C01747=-28.112,-95.435,39.346,-179.6955,-1.2364,-6766.4132
C01748=-32.220,-94.603,39.491,179.9985,-0.0489,-6768.8079
C01749=-36.266,-93.184,39.587,-179.9979,-0.0053,-6771.2653
C01750=-40.247,-91.535,39.587,179.9971,-0.0076,-6773.7346
C01751=-44.111,-89.678,39.491,179.9997,-0.0512,-6776.1917
C01752=-47.604,-87.360,39.346,179.6949,-1.2364,-6778.5867
C01753=-50.060,-84.322,39.203,179.1149,-1.5518,-6780.6966
C01754=-51.116,-81.128,39.027,177.5559,-1.8116,-6782.2136
C01755=-50.704,-78.221,38.697,177.2195,-0.9491,-6782.9519
C01756=-49.835,-75.348,38.031,-179.8330,0.0487,-6783.4806
C01757=-49.130,-72.694,37.169,-173.6149,2.5069,-6784.0527
C01758=-49.058,-70.314,36.333,-164.2153,12.2381,-6784.9034
C01759=-50.194,-67.954,35.726,-167.6473,32.8330,-6786.4513
C01760=-53.078,-65.141,35.484,-177.8974,37.0682,-6789.1737
C01761=-56.256,-62.380,35.473,179.8597,37.2688,-6792.0450
C01762=-59.399,-59.399,35.480,-180.0000,37.2595,-6795.0000
C01763=-62.380,-56.256,35.473,-179.8597,37.2688,-6797.9550
C01764=-65.141,-53.078,35.484,177.8974,37.0682,-6800.8263
C01765=-67.954,-50.194,35.726,167.6473,32.8330,-6803.5487
C01766=-70.314,-49.058,36.333,164.2153,12.2381,-6805.0966
C01767=-72.694,-49.130,37.169,173.6149,2.5069,-6805.9473
C01768=-75.348,-49.835,38.031,179.8330,0.0487,-6806.5194
C01769=-78.221,-50.704,38.697,-177.2195,-0.9491,-6807.0481
C01770=-81.128,-51.116,39.027,-177.5559,-1.8116,-6807.7864
C01771=-84.322,-50.060,39.203,-179.1149,-1.5518,-6809.3034
C01772=-87.360,-47.604,39.346,-179.6949,-1.2364,-6811.4133
C01773=-89.678,-44.111,39.491,-179.9997,-0.0512,-6813.8083
C01774=-91.535,-40.247,39.587,-179.9971,-0.0076,-6816.2654
C01775=-93.184,-36.266,39.587,179.9979,-0.0053,-6818.7347
C01776=-94.603,-32.220,39.491,-179.9985,-0.0489,-6821.1921
C01777=-95.435,-28.112,39.346,179.6955,-1.2364,-6823.5868
C01778=-95.023,-24.227,39.203,179.1127,-1.5540,-6825.6966
C01779=-93.510,-21.221,39.027,177.5538,-1.8150,-6827.2140
C01780=-91.164,-19.458,38.697,177.2185,-0.9486,-6827.9516
C01781=-88.518,-18.041,38.031,-179.8324,0.0477,-6828.4802
C01782=-86.143,-16.662,37.169,-173.6165,2.5084,-6829.0529
C01783=-84.409,-15.030,36.333,-164.2172,12.2420,-6829.9036
C01784=-83.543,-12.558,35.726,-167.6478,32.8316,-6831.4514
C01785=-83.594,-8.530,35.484,-177.9021,37.0692,-6834.1737
C01786=-83.888,-4.330,35.473,179.8571,37.2713,-6837.0452
C01787=-84.003,0.000,35.480,180.0000,37.2584,-6840.0000
C01788=-83.888,4.330,35.473,-179.8571,37.2713,-6842.9548
C01789=-83.594,8.530,35.484,177.8949,37.0687,-6845.8263
C01790=-83.543,12.558,35.726,167.6478,32.8316,-6848.5486
C01791=-84.409,15.030,36.333,164.2172,12.2420,-6850.0964
C01792=-86.143,16.662,37.169,173.6165,2.5084,-6850.9471
C01793=-88.518,18.041,38.031,179.8324,0.0477,-6851.5198
C01794=-91.164,19.458,38.697,-177.2185,-0.9486,-6852.0484
C01795=-93.510,21.221,39.027,-177.5538,-1.8150,-6852.7860
C01796=-95.023,24.227,39.203,-179.1127,-1.5540,-6854.3034
C01797=-95.435,28.112,39.346,-179.6955,-1.2364,-6856.4132
C01798=-94.603,32.220,39.491,179.9985,-0.0489,-6858.8079
C01799=-93.184,36.266,39.587,-179.9979,-0.0053,-6861.2653
C01800=-91.535,40.247,39.587,179.9971,-0.0076,-6863.7346
C01801=-89.678,44.111,39.491,179.9997,-0.0512,-6866.1917
C01802=-87.360,47.604,39.346,179.6949,-1.2364,-6868.5867
C01803=-84.322,50.060,39.203,179.1149,-1.5518,-6870.6966
C01804=-81.128,51.116,39.027,177.5559,-1.8116,-6872.2136
C01805=-78.221,50.704,38.697,177.2195,-0.9491,-6872.9519
C01806=-75.348,49.835,38.031,-179.8330,0.0487,-6873.4806
C01807=-72.694,49.130,37.169,-173.6149,2.5069,-6874.0527
C01808=-70.314,49.058,36.333,-164.2153,12.2381,-6874.9034
C01809=-67.954,50.194,35.726,-167.6473,32.8330,-6876.4513
C01810=-65.141,53.078,35.484,-177.8974,37.0682,-6879.1737
C01811=-62.380,56.256,35.473,179.8597,37.2688,-6882.0450
C01812=-59.399,59.399,35.480,-180.0000,37.2595,-6885.0000
C01813=-56.256,62.380,35.473,-179.8597,37.2688,-6887.9550
C01814=-53.078,65.141,35.484,177.8974,37.0682,-6890.8263
C01815=-50.194,67.954,35.726,167.6473,32.8330,-6893.5487
C01816=-49.058,70.314,36.333,164.2153,12.2381,-6895.0966
C01817=-49.130,72.694,37.169,173.6149,2.5069,-6895.9473
C01818=-49.835,75.348,38.031,179.8330,0.0487,-6896.5194
C01819=-50.704,78.221,38.697,-177.2195,-0.9491,-6897.0481
C01820=-51.116,81.128,39.027,-177.5559,-1.8116,-6897.7864
C01821=-50.060,84.322,39.203,-179.1149,-1.5518,-6899.3034
C01822=-47.604,87.360,39.346,-179.6949,-1.2364,-6901.4133
C01823=-44.111,89.678,39.491,-179.9997,-0.0512,-6903.8083
C01824=-40.247,91.535,39.587,-179.9971,-0.0076,-6906.2654
C01825=-36.266,93.184,39.587,179.9979,-0.0053,-6908.7347
C01826=-32.220,94.603,39.491,-179.9985,-0.0489,-6911.1921
C01827=-28.112,95.435,39.346,179.6955,-1.2364,-6913.5868
C01828=-24.227,95.023,39.203,179.1127,-1.5540,-6915.6966
C01829=-21.221,93.510,39.027,177.5538,-1.8150,-6917.2140
C01830=-19.458,91.164,38.697,177.2185,-0.9486,-6917.9516
C01831=-18.041,88.518,38.031,-179.8324,0.0477,-6918.4802
C01832=-16.662,86.143,37.169,-173.6165,2.5084,-6919.0529
C01833=-15.030,84.409,36.333,-164.2172,12.2420,-6919.9036
C01834=-12.558,83.543,35.726,-167.6478,32.8316,-6921.4514
C01835=-8.530,83.594,35.484,-177.8949,37.0687,-6924.1737
C01836=-4.330,83.888,35.473,179.8571,37.2713,-6927.0452
C01837=0.000,84.003,35.480,-180.0000,37.2584,-6930.0000
C01838=0.000,82.662,37.225,-180.0000,37.7936,-6930.0000
C01839=4.208,82.553,37.217,-179.8407,37.8064,-6932.9180
C01840=8.324,82.270,37.229,177.6416,37.5779,-6935.7775
C01841=12.305,82.260,37.495,166.4964,32.7139,-6938.5076
C01842=14.718,83.232,38.165,164.8382,10.3506,-6940.0280
C01843=16.299,85.134,39.090,174.8249,1.7602,-6940.8382
C01844=17.640,87.735,40.048,-179.1581,-0.2048,-6941.3683
C01845=19.021,90.644,40.789,-176.2692,-1.0819,-6941.8512
C01846=20.743,93.250,41.159,-176.7146,-2.1680,-6942.5410
C01847=23.775,94.968,41.355,-178.8146,-1.9251,-6944.0550
C01848=27.752,95.500,41.515,-179.6323,-1.4088,-6946.2037
C01849=31.992,94.679,41.678,-179.9961,-0.0652,-6948.6701
C01850=36.189,93.214,41.785,179.9967,-0.0074,-6951.2180
C01851=40.323,91.502,41.785,179.9971,-0.0076,-6953.7821
C01852=44.326,89.570,41.678,179.9997,-0.0641,-6956.3297
C01853=47.905,87.153,41.515,179.6318,-1.4120,-6958.7961
C01854=50.341,83.964,41.355,178.8155,-1.9264,-6960.9450
C01855=51.270,80.606,41.159,176.7131,-2.1668,-6962.4587
C01856=50.645,77.545,40.789,176.2678,-1.0827,-6963.1487
C01857=49.565,74.511,40.048,179.1528,-0.2057,-6963.6320
C01858=48.673,71.724,39.090,-174.8246,1.7614,-6964.1614
C01859=48.447,69.261,38.165,-164.8356,10.3507,-6964.9722
C01860=49.465,66.868,37.495,-166.4996,32.7126,-6966.4919
C01861=52.288,64.059,37.229,-177.6432,37.5797,-6969.2230
C01862=55.398,61.349,37.217,179.8424,37.8051,-6972.0820
C01863=58.451,58.451,37.225,-180.0000,37.7926,-6975.0000
C01864=61.349,55.398,37.217,-179.8424,37.8051,-6977.9180
C01865=64.059,52.288,37.229,177.6432,37.5797,-6980.7770
C01866=66.868,49.465,37.495,166.5035,32.7166,-6983.5081
C01867=69.261,48.447,38.165,164.8356,10.3507,-6985.0278
C01868=71.724,48.673,39.090,174.8246,1.7614,-6985.8386
C01869=74.511,49.565,40.048,-179.1528,-0.2057,-6986.3680
C01870=77.545,50.645,40.789,-176.2678,-1.0827,-6986.8513
C01871=80.606,51.270,41.159,-176.7131,-2.1668,-6987.5413
C01872=83.964,50.341,41.355,-178.8155,-1.9264,-6989.0550
C01873=87.153,47.905,41.515,-179.6318,-1.4120,-6991.2039
C01874=89.570,44.326,41.678,-179.9997,-0.0641,-6993.6703
C01875=91.502,40.323,41.785,-179.9971,-0.0076,-6996.2179
C01876=93.214,36.189,41.785,-179.9967,-0.0074,-6998.7820
C01877=94.679,31.992,41.678,179.9961,-0.0652,-7001.3299
C01878=95.500,27.752,41.515,179.6323,-1.4088,-7003.7963
C01879=94.968,23.775,41.355,178.8146,-1.9251,-7005.9450
C01880=93.250,20.743,41.159,176.7146,-2.1680,-7007.4590
C01881=90.644,19.021,40.789,176.2692,-1.0819,-7008.1488
C01882=87.735,17.640,40.048,179.1581,-0.2048,-7008.6317
C01883=85.134,16.299,39.090,-174.8249,1.7602,-7009.1618
C01884=83.232,14.718,38.165,-164.8382,10.3506,-7009.9720
C01885=82.260,12.305,37.495,-166.4964,32.7139,-7011.4924
C01886=82.270,8.324,37.229,-177.6416,37.5779,-7014.2225
C01887=82.553,4.208,37.217,179.8407,37.8064,-7017.0820
C01888=82.662,0.000,37.225,-180.0000,37.7936,-7020.0000
C01889=82.553,-4.208,37.217,-179.8407,37.8064,-7022.9180
C01890=82.270,-8.324,37.229,177.6416,37.5779,-7025.7775
C01891=82.260,-12.305,37.495,166.5029,32.7146,-7028.5076
C01892=83.232,-14.718,38.165,164.8382,10.3506,-7030.0280
C01893=85.134,-16.299,39.090,174.8249,1.7602,-7030.8382
C01894=87.735,-17.640,40.048,-179.1581,-0.2048,-7031.3683
C01895=90.644,-19.021,40.789,-176.2692,-1.0819,-7031.8512
C01896=93.250,-20.743,41.159,-176.7146,-2.1680,-7032.5410
C01897=94.968,-23.775,41.355,-178.8146,-1.9251,-7034.0550
C01898=95.500,-27.752,41.515,-179.6323,-1.4088,-7036.2037
C01899=94.679,-31.992,41.678,-179.9961,-0.0652,-7038.6701
C01900=93.214,-36.189,41.785,179.9967,-0.0074,-7041.2180
C01901=91.502,-40.323,41.785,179.9971,-0.0076,-7043.7821
C01902=89.570,-44.326,41.678,179.9997,-0.0641,-7046.3297
C01903=87.153,-47.905,41.515,179.6318,-1.4120,-7048.7961
C01904=83.964,-50.341,41.355,178.8155,-1.9264,-7050.9450
C01905=80.606,-51.270,41.159,176.7131,-2.1668,-7052.4587
C01906=77.545,-50.645,40.789,176.2678,-1.0827,-7053.1487
C01907=74.511,-49.565,40.048,179.1528,-0.2057,-7053.6320
C01908=71.724,-48.673,39.090,-174.8246,1.7614,-7054.1614
C01909=69.261,-48.447,38.165,-164.8356,10.3507,-7054.9722
C01910=66.868,-49.465,37.495,-166.4996,32.7126,-7056.4919
C01911=64.059,-52.288,37.229,-177.6432,37.5797,-7059.2230
C01912=61.349,-55.398,37.217,179.8424,37.8051,-7062.0820
C01913=58.451,-58.451,37.225,180.0000,37.7926,-7065.0000
C01914=55.398,-61.349,37.217,-179.8424,37.8051,-7067.9180
C01915=52.288,-64.059,37.229,177.6432,37.5797,-7070.7770
C01916=49.465,-66.868,37.495,166.5035,32.7166,-7073.5081
C01917=48.447,-69.261,38.165,164.8356,10.3507,-7075.0278
C01918=48.673,-71.724,39.090,174.8246,1.7614,-7075.8386
C01919=49.565,-74.511,40.048,-179.1528,-0.2057,-7076.3680
C01920=50.645,-77.545,40.789,-176.2678,-1.0827,-7076.8513
C01921=51.270,-80.606,41.159,-176.7131,-2.1668,-7077.5413
C01922=50.341,-83.964,41.355,-178.8155,-1.9264,-7079.0550
C01923=47.905,-87.153,41.515,-179.6318,-1.4120,-7081.2039
C01924=44.326,-89.570,41.678,-179.9997,-0.0641,-7083.6703
C01925=40.323,-91.502,41.785,-179.9971,-0.0076,-7086.2179
C01926=36.189,-93.214,41.785,-179.9967,-0.0074,-7088.7820
C01927=31.992,-94.679,41.678,179.9961,-0.0652,-7091.3299
C01928=27.752,-95.500,41.515,179.6323,-1.4088,-7093.7963
C01929=23.775,-94.968,41.355,178.8146,-1.9251,-7095.9450
C01930=20.743,-93.250,41.159,176.7146,-2.1680,-7097.4590
C01931=19.021,-90.644,40.789,176.2692,-1.0819,-7098.1488
C01932=17.640,-87.735,40.048,179.1581,-0.2048,-7098.6317
C01933=16.299,-85.134,39.090,-174.8249,1.7602,-7099.1618
C01934=14.718,-83.232,38.165,-164.8382,10.3506,-7099.9720
C01935=12.305,-82.260,37.495,-166.4964,32.7139,-7101.4924
C01936=8.324,-82.270,37.229,-177.6416,37.5779,-7104.2225
C01937=4.208,-82.553,37.217,179.8407,37.8064,-7107.0820
C01938=0.000,-82.662,37.225,180.0000,37.7936,-7110.0000
C01939=0.000,-82.662,37.225,180.0000,37.7936,-7110.0000
C01940=-4.208,-82.553,37.217,-179.8407,37.8064,-7112.9180
C01941=-8.324,-82.270,37.229,177.6416,37.5779,-7115.7775
C01942=-12.305,-82.260,37.495,166.5029,32.7146,-7118.5076
C01943=-14.718,-83.232,38.165,164.8382,10.3506,-7120.0280
C01944=-16.299,-85.134,39.090,174.8249,1.7602,-7120.8382
C01945=-17.640,-87.735,40.048,-179.1581,-0.2048,-7121.3683
C01946=-19.021,-90.644,40.789,-176.2692,-1.0819,-7121.8512
C01947=-20.743,-93.250,41.159,-176.7146,-2.1680,-7122.5410
C01948=-23.775,-94.968,41.355,-178.8146,-1.9251,-7124.0550
C01949=-27.752,-95.500,41.515,-179.6323,-1.4088,-7126.2037
C01950=-31.992,-94.679,41.678,-179.9961,-0.0652,-7128.6701
C01951=-36.189,-93.214,41.785,179.9967,-0.0074,-7131.2180
C01952=-40.323,-91.502,41.785,179.9971,-0.0076,-7133.7821
C01953=-44.326,-89.570,41.678,179.9997,-0.0641,-7136.3297
C01954=-47.905,-87.153,41.515,179.6318,-1.4120,-7138.7961
C01955=-50.341,-83.964,41.355,178.8155,-1.9264,-7140.9450
C01956=-51.270,-80.606,41.159,176.7131,-2.1668,-7142.4587
C01957=-50.645,-77.545,40.789,176.2678,-1.0827,-7143.1487
C01958=-49.565,-74.511,40.048,179.1528,-0.2057,-7143.6320
C01959=-48.673,-71.724,39.090,-174.8246,1.7614,-7144.1614
C01960=-48.447,-69.261,38.165,-164.8356,10.3507,-7144.9722
C01961=-49.465,-66.868,37.495,-166.4996,32.7126,-7146.4919
C01962=-52.288,-64.059,37.229,-177.6432,37.5797,-7149.2230
C01963=-55.398,-61.349,37.217,179.8424,37.8051,-7152.0820
C01964=-58.451,-58.451,37.225,-180.0000,37.7926,-7155.0000
C01965=-61.349,-55.398,37.217,-179.8424,37.8051,-7157.9180
C01966=-64.059,-52.288,37.229,177.6432,37.5797,-7160.7770
C01967=-66.868,-49.465,37.495,166.5035,32.7166,-7163.5081
C01968=-69.261,-48.447,38.165,164.8356,10.3507,-7165.0278
C01969=-71.724,-48.673,39.090,174.8246,1.7614,-7165.8386
C01970=-74.511,-49.565,40.048,-179.1528,-0.2057,-7166.3680
C01971=-77.545,-50.645,40.789,-176.2678,-1.0827,-7166.8513
C01972=-80.606,-51.270,41.159,-176.7131,-2.1668,-7167.5413
C01973=-83.964,-50.341,41.355,-178.8155,-1.9264,-7169.0550
C01974=-87.153,-47.905,41.515,-179.6318,-1.4120,-7171.2039
C01975=-89.570,-44.326,41.678,-179.9997,-0.0641,-7173.6703
C01976=-91.502,-40.323,41.785,-179.9971,-0.0076,-7176.2179
C01977=-93.214,-36.189,41.785,-179.9967,-0.0074,-7178.7820
C01978=-94.679,-31.992,41.678,179.9961,-0.0652,-7181.3299
C01979=-95.500,-27.752,41.515,179.6323,-1.4088,-7183.7963
C01980=-94.968,-23.775,41.355,178.8146,-1.9251,-7185.9450
C01981=-93.250,-20.743,41.159,176.7146,-2.1680,-7187.4590
C01982=-90.644,-19.021,40.789,176.2692,-1.0819,-7188.1488
C01983=-87.735,-17.640,40.048,179.1581,-0.2048,-7188.6317
C01984=-85.134,-16.299,39.090,-174.8249,1.7602,-7189.1618
C01985=-83.232,-14.718,38.165,-164.8382,10.3506,-7189.9720
C01986=-82.260,-12.305,37.495,-166.4964,32.7139,-7191.4924
C01987=-82.270,-8.324,37.229,-177.6416,37.5779,-7194.2225
C01988=-82.553,-4.208,37.217,179.8407,37.8064,-7197.0820
C01989=-82.662,0.000,37.225,-180.0000,37.7936,-7200.0000
C01990=-82.553,4.208,37.217,-179.8407,37.8064,-7202.9180
C01991=-82.270,8.324,37.229,177.6416,37.5779,-7205.7775
C01992=-82.260,12.305,37.495,166.5029,32.7146,-7208.5076
C01993=-83.232,14.718,38.165,164.8382,10.3506,-7210.0280
C01994=-85.134,16.299,39.090,174.8249,1.7602,-7210.8382
C01995=-87.735,17.640,40.048,-179.1581,-0.2048,-7211.3683
C01996=-90.644,19.021,40.789,-176.2692,-1.0819,-7211.8512
C01997=-93.250,20.743,41.159,-176.7146,-2.1680,-7212.5410
C01998=-94.968,23.775,41.355,-178.8146,-1.9251,-7214.0550
C01999=-95.500,27.752,41.515,-179.6323,-1.4088,-7216.2037
///TOOL 0
///POSTYPE ANGLE
///ANGLE
EC00000=9.2440,3657.6170
EC00001=6.2165,3658.5035
EC00002=4.0258,3659.6330
EC00003=1.7463,3661.2065
EC00004=0.2718,3663.0322
EC00005=0.0768,3664.8747
EC00006=0.0075,3666.6340
EC00007=0.0074,3668.3657
EC00008=0.0778,3670.1252
EC00009=0.2756,3671.9676
EC00010=1.7445,3673.7937
EC00011=4.0294,3675.3667
EC00012=6.2189,3676.4965
EC00013=9.2462,3677.3831
EC00014=14.9094,3678.2747
EC00015=21.6484,3679.4181
EC00016=25.8724,3681.1629
EC00017=27.0185,3683.8301
EC00018=27.0874,3686.7848
EC00019=27.0775,3690.0000
EC00020=28.8281,3690.0000
EC00021=28.8401,3693.1930
EC00022=28.7637,3696.1402
EC00023=27.4530,3698.8129
EC00024=22.1760,3700.5402
EC00025=14.0567,3701.6582
EC00026=8.0331,3702.5225
EC00027=5.3244,3703.3766
EC00028=3.6143,3704.4702
EC00029=1.5415,3706.0363
EC00030=0.1578,3707.8866
EC00031=0.0671,3709.7782
EC00032=0.0053,3711.6011
EC00033=0.0075,3713.3991
EC00034=0.0692,3715.2213
EC00035=0.1565,3717.1138
EC00036=1.5379,3718.9637
EC00037=3.6128,3720.5297
EC00038=5.3283,3721.6234
EC00039=8.0333,3722.4779
EC00040=14.0579,3723.3415
EC00041=22.1779,3724.4600
EC00042=27.4539,3726.1873
EC00043=28.7627,3728.8598
EC00044=28.8407,3731.8071
EC00045=28.8305,3735.0000
EC00046=28.8407,3738.1929
EC00047=28.7627,3741.1402
EC00048=27.4539,3743.8127
EC00049=22.1779,3745.5400
EC00050=14.0579,3746.6585
EC00051=8.0333,3747.5221
EC00052=5.3283,3748.3766
EC00053=3.6128,3749.4703
EC00054=1.5379,3751.0363
EC00055=0.1565,3752.8862
EC00056=0.0692,3754.7787
EC00057=0.0075,3756.6009
EC00058=0.0053,3758.3989
EC00059=0.0671,3760.2218
EC00060=0.1578,3762.1134
EC00061=1.5415,3763.9637
EC00062=3.6143,3765.5298
EC00063=5.3244,3766.6234
EC00064=8.0331,3767.4775
EC00065=14.0567,3768.3418
EC00066=22.1760,3769.4598
EC00067=27.4530,3771.1871
EC00068=28.7637,3773.8598
EC00069=28.8401,3776.8070
EC00070=28.8281,3780.0000
EC00071=28.8401,3783.1930
EC00072=28.7637,3786.1402
EC00073=27.4530,3788.8128
EC00074=22.1760,3790.5402
EC00075=14.0567,3791.6582
EC00076=8.0331,3792.5225
EC00077=5.3244,3793.3766
EC00078=3.6143,3794.4702
EC00079=1.5415,3796.0363
EC00080=0.1578,3797.8866
EC00081=0.0671,3799.7782
EC00082=0.0053,3801.6011
EC00083=0.0075,3803.3991
EC00084=0.0692,3805.2213
EC00085=0.1565,3807.1138
EC00086=1.5379,3808.9637
EC00087=3.6128,3810.5297
EC00088=5.3283,3811.6234
EC00089=8.0333,3812.4779
EC00090=14.0579,3813.3415
EC00091=22.1779,3814.4600
EC00092=27.4539,3816.1873
EC00093=28.7627,3818.8598
EC00094=28.8407,3821.8071
EC00095=28.8305,3825.0000
EC00096=28.8407,3828.1929
EC00097=28.7627,3831.1402
EC00098=27.4539,3833.8127
EC00099=22.1779,3835.5400
EC00100=14.0579,3836.6585
EC00101=8.0333,3837.5221
EC00102=5.3283,3838.3766
EC00103=3.6128,3839.4703
EC00104=1.5379,3841.0363
EC00105=0.1565,3842.8862
EC00106=0.0692,3844.7787
EC00107=0.0075,3846.6009
EC00108=0.0053,3848.3989
EC00109=0.0671,3850.2218
EC00110=0.1578,3852.1134
EC00111=1.5415,3853.9637
EC00112=3.6143,3855.5298
EC00113=5.3244,3856.6234
EC00114=8.0331,3857.4775
EC00115=14.0567,3858.3418
EC00116=22.1760,3859.4598
EC00117=27.4530,3861.1871
EC00118=28.7637,3863.8598
EC00119=28.8401,3866.8070
EC00120=28.8281,3870.0000
EC00121=28.8281,3870.0000
EC00122=28.8401,3873.1930
EC00123=28.7637,3876.1402
EC00124=27.4530,3878.8128
EC00125=22.1760,3880.5402
EC00126=14.0567,3881.6582
EC00127=8.0331,3882.5225
EC00128=5.3244,3883.3766
EC00129=3.6143,3884.4702
EC00130=1.5415,3886.0363
EC00131=0.1578,3887.8866
EC00132=0.0671,3889.7782
EC00133=0.0053,3891.6011
EC00134=0.0075,3893.3991
EC00135=0.0692,3895.2213
EC00136=0.1565,3897.1138
EC00137=1.5379,3898.9637
EC00138=3.6128,3900.5297
EC00139=5.3283,3901.6234
EC00140=8.0333,3902.4779
EC00141=14.0579,3903.3415
EC00142=22.1779,3904.4600
EC00143=27.4539,3906.1873
EC00144=28.7627,3908.8598
EC00145=28.8407,3911.8071
EC00146=28.8305,3915.0000
EC00147=28.8407,3918.1929
EC00148=28.7627,3921.1402
EC00149=27.4539,3923.8127
EC00150=22.1779,3925.5400
EC00151=14.0579,3926.6585
EC00152=8.0333,3927.5221
EC00153=5.3283,3928.3766
EC00154=3.6128,3929.4703
EC00155=1.5379,3931.0363
EC00156=0.1565,3932.8862
EC00157=0.0692,3934.7787
EC00158=0.0075,3936.6009
EC00159=0.0053,3938.3989
EC00160=0.0671,3940.2218
EC00161=0.1578,3942.1134
EC00162=1.5415,3943.9637
EC00163=3.6143,3945.5298
EC00164=5.3244,3946.6234
EC00165=8.0331,3947.4775
EC00166=14.0567,3948.3418
EC00167=22.1760,3949.4598
EC00168=27.4530,3951.1871
EC00169=28.7637,3953.8598
EC00170=28.8401,3956.8070
EC00171=28.8281,3960.0000
EC00172=28.8401,3963.1930
EC00173=28.7637,3966.1402
EC00174=27.4530,3968.8128
EC00175=22.1760,3970.5402
EC00176=14.0567,3971.6582
EC00177=8.0331,3972.5225
EC00178=5.3244,3973.3766
EC00179=3.6143,3974.4702
EC00180=1.5415,3976.0363
EC00181=0.1578,3977.8866
EC00182=0.0671,3979.7782
EC00183=0.0053,3981.6011
EC00184=0.0075,3983.3991
EC00185=0.0692,3985.2213
EC00186=0.1565,3987.1138
EC00187=1.5379,3988.9637
EC00188=3.6128,3990.5297
EC00189=5.3283,3991.6234
EC00190=8.0333,3992.4779
EC00191=14.0579,3993.3415
EC00192=22.1779,3994.4600
EC00193=27.4539,3996.1873
EC00194=28.7627,3998.8598
EC00195=28.8407,4001.8071
EC00196=28.8305,4005.0000
EC00197=28.8407,4008.1929
EC00198=28.7627,4011.1402
EC00199=27.4539,4013.8127
EC00200=22.1779,4015.5400
EC00201=14.0579,4016.6585
EC00202=8.0333,4017.5221
EC00203=5.3283,4018.3766
EC00204=3.6128,4019.4703
EC00205=1.5379,4021.0363
EC00206=0.1565,4022.8862
EC00207=0.0692,4024.7787
EC00208=0.0075,4026.6009
EC00209=0.0053,4028.3989
EC00210=0.0671,4030.2218
EC00211=0.1578,4032.1134
EC00212=1.5415,4033.9637
EC00213=3.6143,4035.5298
EC00214=5.3244,4036.6234
EC00215=8.0331,4037.4775
EC00216=14.0567,4038.3418
EC00217=22.1760,4039.4598
EC00218=27.4530,4041.1872
EC00219=28.7637,4043.8598
EC00220=28.8401,4046.8070
EC00221=28.8281,4050.0000
EC00222=30.3909,4050.0000
EC00223=30.3994,4053.1693
EC00224=30.3134,4056.1086
EC00225=28.8062,4058.7858
EC00226=22.2216,4060.4951
EC00227=12.7358,4061.5862
EC00228=6.5920,4062.4199
EC00229=4.2313,4063.2394
EC00230=3.0336,4064.2944
EC00231=1.2647,4065.8535
EC00232=0.0236,4067.7299
EC00233=0.0597,4069.6757
EC00234=0.0053,4071.5655
EC00235=0.0053,4073.4348
EC00236=0.0564,4075.3246
EC00237=0.0205,4077.2701
EC00238=1.2668,4079.1464
EC00239=3.0331,4080.7059
EC00240=4.2307,4081.7605
EC00241=6.5908,4082.5800
EC00242=12.7370,4083.4139
EC00243=22.2236,4084.5045
EC00244=28.8036,4086.2144
EC00245=30.3167,4088.8913
EC00246=30.4010,4091.8309
EC00247=30.3891,4095.0000
EC00248=30.4010,4098.1691
EC00249=30.3167,4101.1087
EC00250=28.8076,4103.7856
EC00251=22.2236,4105.4955
EC00252=12.7370,4106.5861
EC00253=6.5908,4107.4200
EC00254=4.2307,4108.2395
EC00255=3.0331,4109.2941
EC00256=1.2668,4110.8536
EC00257=0.0205,4112.7299
EC00258=0.0564,4114.6754
EC00259=0.0053,4116.5652
EC00260=0.0053,4118.4345
EC00261=0.0597,4120.3243
EC00262=0.0236,4122.2701
EC00263=1.2647,4124.1465
EC00264=3.0336,4125.7056
EC00265=4.2313,4126.7606
EC00266=6.5920,4127.5801
EC00267=12.7358,4128.4138
EC00268=22.2216,4129.5049
EC00269=28.8062,4131.2142
EC00270=30.3134,4133.8914
EC00271=30.3994,4136.8307
EC00272=30.3909,4140.0000
EC00273=30.3994,4143.1693
EC00274=30.3134,4146.1086
EC00275=28.8062,4148.7858
EC00276=22.2216,4150.4951
EC00277=12.7358,4151.5862
EC00278=6.5920,4152.4199
EC00279=4.2313,4153.2394
EC00280=3.0336,4154.2944
EC00281=1.2647,4155.8535
EC00282=0.0236,4157.7299
EC00283=0.0597,4159.6757
EC00284=0.0053,4161.5655
EC00285=0.0053,4163.4348
EC00286=0.0564,4165.3246
EC00287=0.0205,4167.2701
EC00288=1.2668,4169.1464
EC00289=3.0331,4170.7059
EC00290=4.2307,4171.7605
EC00291=6.5908,4172.5800
EC00292=12.7370,4173.4139
EC00293=22.2236,4174.5045
EC00294=28.8036,4176.2144
EC00295=30.3167,4178.8913
EC00296=30.4010,4181.8309
EC00297=30.3891,4185.0000
EC00298=30.4010,4188.1691
EC00299=30.3167,4191.1087
EC00300=28.8076,4193.7856
EC00301=22.2236,4195.4955
EC00302=12.7370,4196.5861
EC00303=6.5908,4197.4200
EC00304=4.2307,4198.2395
EC00305=3.0331,4199.2941
EC00306=1.2668,4200.8536
EC00307=0.0205,4202.7299
EC00308=0.0564,4204.6754
EC00309=0.0053,4206.5652
EC00310=0.0053,4208.4345
EC00311=0.0597,4210.3243
EC00312=0.0236,4212.2701
EC00313=1.2647,4214.1465
EC00314=3.0336,4215.7056
EC00315=4.2313,4216.7606
EC00316=6.5920,4217.5801
EC00317=12.7358,4218.4138
EC00318=22.2216,4219.5049
EC00319=28.8062,4221.2142
EC00320=30.3134,4223.8914
EC00321=30.3994,4226.8307
EC00322=30.3909,4230.0000
EC00323=30.3909,4230.0000
EC00324=30.3994,4233.1693
EC00325=30.3134,4236.1086
EC00326=28.8062,4238.7858
EC00327=22.2216,4240.4951
EC00328=12.7358,4241.5862
EC00329=6.5920,4242.4199
EC00330=4.2313,4243.2394
EC00331=3.0336,4244.2944
EC00332=1.2647,4245.8535
EC00333=0.0236,4247.7299
EC00334=0.0597,4249.6757
EC00335=0.0053,4251.5655
EC00336=0.0053,4253.4348
EC00337=0.0564,4255.3246
EC00338=0.0205,4257.2701
EC00339=1.2668,4259.1464
EC00340=3.0331,4260.7059
EC00341=4.2307,4261.7605
EC00342=6.5908,4262.5800
EC00343=12.7370,4263.4139
EC00344=22.2236,4264.5045
EC00345=28.8036,4266.2144
EC00346=30.3167,4268.8913
EC00347=30.4010,4271.8309
EC00348=30.3891,4275.0000
EC00349=30.4010,4278.1691
EC00350=30.3167,4281.1087
EC00351=28.8076,4283.7856
EC00352=22.2236,4285.4955
EC00353=12.7370,4286.5861
EC00354=6.5908,4287.4200
EC00355=4.2307,4288.2395
EC00356=3.0331,4289.2941
EC00357=1.2668,4290.8536
EC00358=0.0205,4292.7299
EC00359=0.0564,4294.6754
EC00360=0.0053,4296.5652
EC00361=0.0053,4298.4345
EC00362=0.0597,4300.3243
EC00363=0.0236,4302.2701
EC00364=1.2647,4304.1465
EC00365=3.0336,4305.7056
EC00366=4.2313,4306.7606
EC00367=6.5920,4307.5801
EC00368=12.7358,4308.4138
EC00369=22.2216,4309.5049
EC00370=28.8062,4311.2142
EC00371=30.3134,4313.8914
EC00372=30.3994,4316.8307
EC00373=30.3909,4320.0000
EC00374=30.3994,4323.1693
EC00375=30.3134,4326.1086
EC00376=28.8062,4328.7858
EC00377=22.2216,4330.4951
EC00378=12.7358,4331.5862
EC00379=6.5920,4332.4199
EC00380=4.2313,4333.2394
EC00381=3.0336,4334.2944
EC00382=1.2647,4335.8535
EC00383=0.0236,4337.7299
EC00384=0.0597,4339.6757
EC00385=0.0053,4341.5655
EC00386=0.0053,4343.4348
EC00387=0.0564,4345.3246
EC00388=0.0205,4347.2701
EC00389=1.2668,4349.1464
EC00390=3.0331,4350.7059
EC00391=4.2307,4351.7605
EC00392=6.5908,4352.5800
EC00393=12.7370,4353.4139
EC00394=22.2236,4354.5045
EC00395=28.8036,4356.2144
EC00396=30.3167,4358.8913
EC00397=30.4010,4361.8309
EC00398=30.3891,4365.0000
EC00399=30.4010,4368.1691
EC00400=30.3167,4371.1087
EC00401=28.8076,4373.7856
EC00402=22.2236,4375.4955
EC00403=12.7370,4376.5861
EC00404=6.5908,4377.4200
EC00405=4.2307,4378.2395
EC00406=3.0331,4379.2941
EC00407=1.2668,4380.8536
EC00408=0.0205,4382.7299
EC00409=0.0564,4384.6754
EC00410=0.0053,4386.5652
EC00411=0.0053,4388.4345
EC00412=0.0597,4390.3243
EC00413=0.0236,4392.2701
EC00414=1.2647,4394.1465
EC00415=3.0336,4395.7056
EC00416=4.2313,4396.7606
EC00417=6.5920,4397.5801
EC00418=12.7358,4398.4138
EC00419=22.2216,4399.5049
EC00420=28.8062,4401.2142
EC00421=30.3134,4403.8914
EC00422=30.3994,4406.8307
EC00423=30.3909,4410.0000
EC00424=31.7764,4410.0000
EC00425=31.7913,4413.1434
EC00426=31.6940,4416.0750
EC00427=29.9498,4418.7577
EC00428=21.7872,4420.4474
EC00429=11.0995,4421.5089
EC00430=5.1205,4422.3101
EC00431=3.0731,4423.0930
EC00432=2.3162,4424.1066
EC00433=0.9262,4425.6587
EC00434=-0.1326,4427.5637
EC00435=0.0435,4429.5659
EC00436=0.0053,4431.5274
EC00437=0.0053,4433.4725
EC00438=0.0436,4435.4343
EC00439=-0.1336,4437.4359
EC00440=0.9269,4439.3411
EC00441=2.3167,4440.8935
EC00442=3.0727,4441.9071
EC00443=5.1213,4442.6899
EC00444=11.0962,4443.4910
EC00445=21.7869,4444.5530
EC00446=29.9481,4446.2423
EC00447=31.6931,4448.9252
EC00448=31.7887,4451.8567
EC00449=31.7790,4455.0000
EC00450=31.7887,4458.1433
EC00451=31.6931,4461.0748
EC00452=29.9481,4463.7577
EC00453=21.7869,4465.4470
EC00454=11.0962,4466.5090
EC00455=5.1213,4467.3101
EC00456=3.0727,4468.0929
EC00457=2.3167,4469.1065
EC00458=0.9269,4470.6589
EC00459=-0.1336,4472.5641
EC00460=0.0436,4474.5657
EC00461=0.0053,4476.5275
EC00462=0.0053,4478.4726
EC00463=0.0435,4480.4341
EC00464=-0.1326,4482.4363
EC00465=0.9262,4484.3413
EC00466=2.3162,4485.8934
EC00467=3.0731,4486.9070
EC00468=5.1205,4487.6899
EC00469=11.0995,4488.4911
EC00470=21.7872,4489.5526
EC00471=29.9498,4491.2423
EC00472=31.6940,4493.9250
EC00473=31.7913,4496.8566
EC00474=31.7764,4500.0000
EC00475=31.7913,4503.1434
EC00476=31.6940,4506.0750
EC00477=29.9498,4508.7577
EC00478=21.7872,4510.4474
EC00479=11.0995,4511.5089
EC00480=5.1205,4512.3101
EC00481=3.0731,4513.0930
EC00482=2.3162,4514.1066
EC00483=0.9262,4515.6587
EC00484=-0.1326,4517.5637
EC00485=0.0435,4519.5659
EC00486=0.0053,4521.5274
EC00487=0.0053,4523.4725
EC00488=0.0436,4525.4343
EC00489=-0.1336,4527.4359
EC00490=0.9269,4529.3411
EC00491=2.3167,4530.8935
EC00492=3.0727,4531.9071
EC00493=5.1213,4532.6899
EC00494=11.0962,4533.4910
EC00495=21.7869,4534.5530
EC00496=29.9481,4536.2423
EC00497=31.6931,4538.9252
EC00498=31.7887,4541.8567
EC00499=31.7790,4545.0000
EC00500=31.7887,4548.1433
EC00501=31.6931,4551.0748
EC00502=29.9481,4553.7577
EC00503=21.7869,4555.4470
EC00504=11.0962,4556.5090
EC00505=5.1213,4557.3101
EC00506=3.0727,4558.0929
EC00507=2.3167,4559.1065
EC00508=0.9269,4560.6589
EC00509=-0.1336,4562.5641
EC00510=0.0436,4564.5657
EC00511=0.0053,4566.5275
EC00512=0.0053,4568.4726
EC00513=0.0435,4570.4341
EC00514=-0.1326,4572.4363
EC00515=0.9262,4574.3413
EC00516=2.3162,4575.8934
EC00517=3.0731,4576.9070
EC00518=5.1205,4577.6899
EC00519=11.0995,4578.4911
EC00520=21.7872,4579.5526
EC00521=29.9498,4581.2423
EC00522=31.6940,4583.9250
EC00523=31.7913,4586.8566
EC00524=31.7764,4590.0000
EC00525=31.7764,4590.0000
EC00526=31.7913,4593.1434
EC00527=31.6940,4596.0750
EC00528=29.9498,4598.7577
EC00529=21.7872,4600.4474
EC00530=11.0995,4601.5089
EC00531=5.1205,4602.3101
EC00532=3.0731,4603.0930
EC00533=2.3162,4604.1066
EC00534=0.9262,4605.6587
EC00535=-0.1326,4607.5637
EC00536=0.0435,4609.5659
EC00537=0.0053,4611.5274
EC00538=0.0053,4613.4725
EC00539=0.0436,4615.4343
EC00540=-0.1336,4617.4359
EC00541=0.9269,4619.3411
EC00542=2.3167,4620.8935
EC00543=3.0727,4621.9071
EC00544=5.1213,4622.6899
EC00545=11.0962,4623.4910
EC00546=21.7869,4624.5530
EC00547=29.9481,4626.2423
EC00548=31.6931,4628.9252
EC00549=31.7887,4631.8567
EC00550=31.7790,4635.0000
EC00551=31.7887,4638.1433
EC00552=31.6931,4641.0748
EC00553=29.9481,4643.7577
EC00554=21.7869,4645.4470
EC00555=11.0962,4646.5090
EC00556=5.1213,4647.3101
EC00557=3.0727,4648.0929
EC00558=2.3167,4649.1065
EC00559=0.9269,4650.6589
EC00560=-0.1336,4652.5641
EC00561=0.0436,4654.5657
EC00562=0.0053,4656.5275
EC00563=0.0053,4658.4726
EC00564=0.0435,4660.4341
EC00565=-0.1326,4662.4363
EC00566=0.9262,4664.3413
EC00567=2.3162,4665.8934
EC00568=3.0731,4666.9070
EC00569=5.1205,4667.6899
EC00570=11.0995,4668.4911
EC00571=21.7872,4669.5526
EC00572=29.9498,4671.2423
EC00573=31.6940,4673.9250
EC00574=31.7913,4676.8566
EC00575=31.7764,4680.0000
EC00576=31.7913,4683.1434
EC00577=31.6940,4686.0750
EC00578=29.9498,4688.7577
EC00579=21.7872,4690.4474
EC00580=11.0995,4691.5089
EC00581=5.1205,4692.3101
EC00582=3.0731,4693.0930
EC00583=2.3162,4694.1066
EC00584=0.9262,4695.6587
EC00585=-0.1326,4697.5637
EC00586=0.0435,4699.5659
EC00587=0.0053,4701.5274
EC00588=0.0053,4703.4725
EC00589=0.0436,4705.4343
EC00590=-0.1336,4707.4359
EC00591=0.9269,4709.3411
EC00592=2.3167,4710.8935
EC00593=3.0727,4711.9071
EC00594=5.1213,4712.6899
EC00595=11.0962,4713.4910
EC00596=21.7869,4714.5530
EC00597=29.9481,4716.2423
EC00598=31.6931,4718.9252
EC00599=31.7887,4721.8567
EC00600=31.7790,4725.0000
EC00601=31.7887,4728.1433
EC00602=31.6931,4731.0748
EC00603=29.9481,4733.7577
EC00604=21.7869,4735.4470
EC00605=11.0962,4736.5090
EC00606=5.1213,4737.3101
EC00607=3.0727,4738.0929
EC00608=2.3167,4739.1065
EC00609=0.9269,4740.6589
EC00610=-0.1336,4742.5641
EC00611=0.0436,4744.5657
EC00612=0.0053,4746.5275
EC00613=0.0053,4748.4726
EC00614=0.0435,4750.4341
EC00615=-0.1326,4752.4363
EC00616=0.9262,4754.3413
EC00617=2.3162,4755.8934
EC00618=3.0731,4756.9070
EC00619=5.1205,4757.6899
EC00620=11.0995,4758.4911
EC00621=21.7872,4759.5526
EC00622=29.9498,4761.2423
EC00623=31.6940,4763.9250
EC00624=31.7913,4766.8566
EC00625=31.7764,4770.0000
EC00626=33.0099,4770.0000
EC00627=33.0210,4773.1159
EC00628=32.9112,4776.0385
EC00629=30.8885,4778.7274
EC00630=20.8945,4780.3963
EC00631=9.3354,4781.4267
EC00632=3.7616,4782.1938
EC00633=1.9745,4782.9380
EC00634=1.5285,4783.9087
EC00635=0.5486,4785.4538
EC00636=-0.3035,4787.3887
EC00637=0.0308,4789.4506
EC00638=0.0000,4791.4875
EC00639=0.0000,4793.5125
EC00640=0.0308,4795.5494
EC00641=-0.3033,4797.6113
EC00642=0.5487,4799.5463
EC00643=1.5238,4801.0916
EC00644=1.9748,4802.0621
EC00645=3.7642,4802.8061
EC00646=9.3352,4803.5730
EC00647=20.8949,4804.6038
EC00648=30.8897,4806.2732
EC00649=32.9101,4808.9613
EC00650=33.0184,4811.8843
EC00651=33.0078,4815.0000
EC00652=33.0184,4818.1157
EC00653=32.9101,4821.0387
EC00654=30.8897,4823.7268
EC00655=20.8949,4825.3962
EC00656=9.3352,4826.4270
EC00657=3.7642,4827.1939
EC00658=1.9748,4827.9379
EC00659=1.5238,4828.9084
EC00660=0.5487,4830.4537
EC00661=-0.3033,4832.3887
EC00662=0.0308,4834.4506
EC00663=0.0000,4836.4875
EC00664=0.0000,4838.5125
EC00665=0.0308,4840.5494
EC00666=-0.3035,4842.6113
EC00667=0.5486,4844.5462
EC00668=1.5285,4846.0913
EC00669=1.9745,4847.0620
EC00670=3.7616,4847.8062
EC00671=9.3354,4848.5733
EC00672=20.8945,4849.6037
EC00673=30.8885,4851.2726
EC00674=32.9112,4853.9615
EC00675=33.0210,4856.8841
EC00676=33.0099,4860.0000
EC00677=33.0210,4863.1159
EC00678=32.9112,4866.0385
EC00679=30.8885,4868.7274
EC00680=20.8945,4870.3963
EC00681=9.3354,4871.4267
EC00682=3.7616,4872.1938
EC00683=1.9745,4872.9380
EC00684=1.5285,4873.9087
EC00685=0.5486,4875.4538
EC00686=-0.3035,4877.3887
EC00687=0.0308,4879.4506
EC00688=0.0000,4881.4875
EC00689=0.0000,4883.5125
EC00690=0.0308,4885.5494
EC00691=-0.3033,4887.6113
EC00692=0.5487,4889.5463
EC00693=1.5238,4891.0916
EC00694=1.9748,4892.0621
EC00695=3.7642,4892.8061
EC00696=9.3352,4893.5730
EC00697=20.8949,4894.6038
EC00698=30.8897,4896.2732
EC00699=32.9101,4898.9613
EC00700=33.0184,4901.8843
EC00701=33.0078,4905.0000
EC00702=33.0184,4908.1157
EC00703=32.9101,4911.0387
EC00704=30.8897,4913.7268
EC00705=20.8949,4915.3962
EC00706=9.3352,4916.4270
EC00707=3.7642,4917.1939
EC00708=1.9748,4917.9379
EC00709=1.5238,4918.9084
EC00710=0.5487,4920.4537
EC00711=-0.3033,4922.3887
EC00712=0.0308,4924.4506
EC00713=0.0000,4926.4875
EC00714=0.0000,4928.5125
EC00715=0.0308,4930.5494
EC00716=-0.3035,4932.6113
EC00717=0.5486,4934.5462
EC00718=1.5285,4936.0913
EC00719=1.9745,4937.0620
EC00720=3.7616,4937.8062
EC00721=9.3354,4938.5733
EC00722=20.8945,4939.6037
EC00723=30.8885,4941.2726
EC00724=32.9112,4943.9615
EC00725=33.0210,4946.8841
EC00726=33.0099,4950.0000
EC00727=33.0099,4950.0000
EC00728=33.0210,4953.1159
EC00729=32.9112,4956.0385
EC00730=30.8885,4958.7274
EC00731=20.8945,4960.3963
EC00732=9.3354,4961.4267
EC00733=3.7616,4962.1938
EC00734=1.9745,4962.9380
EC00735=1.5285,4963.9087
EC00736=0.5486,4965.4538
EC00737=-0.3035,4967.3887
EC00738=0.0308,4969.4506
EC00739=0.0000,4971.4875
EC00740=0.0000,4973.5125
EC00741=0.0308,4975.5494
EC00742=-0.3033,4977.6113
EC00743=0.5487,4979.5463
EC00744=1.5238,4981.0916
EC00745=1.9748,4982.0621
EC00746=3.7642,4982.8061
EC00747=9.3352,4983.5730
EC00748=20.8949,4984.6038
EC00749=30.8897,4986.2732
EC00750=32.9101,4988.9613
EC00751=33.0184,4991.8843
EC00752=33.0078,4995.0000
EC00753=33.0184,4998.1157
EC00754=32.9101,5001.0387
EC00755=30.8897,5003.7268
EC00756=20.8949,5005.3962
EC00757=9.3352,5006.4270
EC00758=3.7642,5007.1939
EC00759=1.9748,5007.9379
EC00760=1.5238,5008.9084
EC00761=0.5487,5010.4537
EC00762=-0.3033,5012.3887
EC00763=0.0308,5014.4506
EC00764=0.0000,5016.4875
EC00765=0.0000,5018.5125
EC00766=0.0308,5020.5494
EC00767=-0.3035,5022.6113
EC00768=0.5486,5024.5462
EC00769=1.5285,5026.0913
EC00770=1.9745,5027.0620
EC00771=3.7616,5027.8062
EC00772=9.3354,5028.5733
EC00773=20.8945,5029.6037
EC00774=30.8885,5031.2726
EC00775=32.9112,5033.9615
EC00776=33.0210,5036.8841
EC00777=33.0099,5040.0000
EC00778=33.0210,5043.1159
EC00779=32.9112,5046.0385
EC00780=30.8885,5048.7274
EC00781=20.8945,5050.3963
EC00782=9.3354,5051.4267
EC00783=3.7616,5052.1938
EC00784=1.9745,5052.9380
EC00785=1.5285,5053.9087
EC00786=0.5486,5055.4538
EC00787=-0.3035,5057.3887
EC00788=0.0308,5059.4506
EC00789=0.0000,5061.4875
EC00790=0.0000,5063.5125
EC00791=0.0308,5065.5494
EC00792=-0.3033,5067.6113
EC00793=0.5487,5069.5463
EC00794=1.5238,5071.0916
EC00795=1.9748,5072.0621
EC00796=3.7642,5072.8061
EC00797=9.3352,5073.5730
EC00798=20.8949,5074.6038
EC00799=30.8897,5076.2732
EC00800=32.9101,5078.9613
EC00801=33.0184,5081.8843
EC00802=33.0078,5085.0000
EC00803=33.0184,5088.1157
EC00804=32.9101,5091.0387
EC00805=30.8897,5093.7268
EC00806=20.8949,5095.3962
EC00807=9.3352,5096.4270
EC00808=3.7642,5097.1939
EC00809=1.9748,5097.9379
EC00810=1.5238,5098.9084
EC00811=0.5487,5100.4537
EC00812=-0.3033,5102.3887
EC00813=0.0308,5104.4506
EC00814=0.0000,5106.4875
EC00815=0.0000,5108.5125
EC00816=0.0308,5110.5494
EC00817=-0.3035,5112.6113
EC00818=0.5486,5114.5462
EC00819=1.5285,5116.0913
EC00820=1.9745,5117.0620
EC00821=3.7616,5117.8062
EC00822=9.3354,5118.5733
EC00823=20.8945,5119.6037
EC00824=30.8885,5121.2726
EC00825=32.9112,5123.9615
EC00826=33.0210,5126.8841
EC00827=33.0099,5130.0000
EC00828=34.0969,5130.0000
EC00829=34.1086,5133.0871
EC00830=33.9818,5136.0002
EC00831=31.6332,5138.6952
EC00832=19.6025,5140.3419
EC00833=7.5978,5141.3400
EC00834=2.6020,5142.0705
EC00835=1.0211,5142.7745
EC00836=0.7176,5143.7009
EC00837=0.1337,5145.2391
EC00838=-0.4893,5147.2060
EC00839=0.0181,5149.3299
EC00840=0.0000,5151.4458
EC00841=0.0000,5153.5540
EC00842=0.0128,5155.6698
EC00843=-0.4862,5157.7938
EC00844=0.1365,5159.7609
EC00845=0.7177,5161.2994
EC00846=1.0199,5162.2255
EC00847=2.6033,5162.9290
EC00848=7.5993,5163.6599
EC00849=19.5985,5164.6583
EC00850=31.6349,5166.3048
EC00851=33.9827,5168.9993
EC00852=34.1079,5171.9128
EC00853=34.0966,5175.0000
EC00854=34.1079,5178.0872
EC00855=33.9827,5181.0007
EC00856=31.6349,5183.6952
EC00857=19.5985,5185.3417
EC00858=7.5993,5186.3401
EC00859=2.6033,5187.0710
EC00860=1.0199,5187.7745
EC00861=0.7177,5188.7006
EC00862=0.1365,5190.2391
EC00863=-0.4862,5192.2062
EC00864=0.0128,5194.3302
EC00865=0.0000,5196.4460
EC00866=0.0000,5198.5542
EC00867=0.0181,5200.6701
EC00868=-0.4893,5202.7940
EC00869=0.1337,5204.7609
EC00870=0.7176,5206.2991
EC00871=1.0211,5207.2255
EC00872=2.6020,5207.9295
EC00873=7.5978,5208.6600
EC00874=19.6025,5209.6581
EC00875=31.6332,5211.3048
EC00876=33.9818,5213.9998
EC00877=34.1086,5216.9129
EC00878=34.0969,5220.0000
EC00879=34.1086,5223.0871
EC00880=33.9818,5226.0002
EC00881=31.6332,5228.6952
EC00882=19.6025,5230.3419
EC00883=7.5978,5231.3400
EC00884=2.6020,5232.0705
EC00885=1.0211,5232.7745
EC00886=0.7176,5233.7009
EC00887=0.1337,5235.2391
EC00888=-0.4893,5237.2060
EC00889=0.0181,5239.3299
EC00890=0.0000,5241.4458
EC00891=0.0000,5243.5540
EC00892=0.0128,5245.6698
EC00893=-0.4862,5247.7938
EC00894=0.1365,5249.7609
EC00895=0.7177,5251.2994
EC00896=1.0199,5252.2255
EC00897=2.6033,5252.9290
EC00898=7.5993,5253.6599
EC00899=19.5985,5254.6583
EC00900=31.6349,5256.3048
EC00901=33.9827,5258.9993
EC00902=34.1079,5261.9128
EC00903=34.0966,5265.0000
EC00904=34.1079,5268.0872
EC00905=33.9827,5271.0007
EC00906=31.6349,5273.6952
EC00907=19.5985,5275.3417
EC00908=7.5993,5276.3401
EC00909=2.6033,5277.0710
EC00910=1.0199,5277.7745
EC00911=0.7177,5278.7006
EC00912=0.1365,5280.2391
EC00913=-0.4862,5282.2062
EC00914=0.0128,5284.3302
EC00915=0.0000,5286.4460
EC00916=0.0000,5288.5542
EC00917=0.0181,5290.6701
EC00918=-0.4893,5292.7940
EC00919=0.1337,5294.7609
EC00920=0.7176,5296.2991
EC00921=1.0211,5297.2255
EC00922=2.6020,5297.9295
EC00923=7.5978,5298.6600
EC00924=19.6025,5299.6581
EC00925=31.6332,5301.3048
EC00926=33.9818,5303.9998
EC00927=34.1086,5306.9129
EC00928=34.0969,5310.0000
EC00929=34.0969,5310.0000
EC00930=34.1086,5313.0871
EC00931=33.9818,5316.0002
EC00932=31.6332,5318.6952
EC00933=19.6025,5320.3419
EC00934=7.5978,5321.3400
EC00935=2.6020,5322.0705
EC00936=1.0211,5322.7745
EC00937=0.7176,5323.7009
EC00938=0.1337,5325.2391
EC00939=-0.4893,5327.2060
EC00940=0.0181,5329.3299
EC00941=0.0000,5331.4458
EC00942=0.0000,5333.5540
EC00943=0.0128,5335.6698
EC00944=-0.4862,5337.7938
EC00945=0.1365,5339.7609
EC00946=0.7177,5341.2994
EC00947=1.0199,5342.2255
EC00948=2.6033,5342.9290
EC00949=7.5993,5343.6599
EC00950=19.5985,5344.6583
EC00951=31.6349,5346.3048
EC00952=33.9827,5348.9993
EC00953=34.1079,5351.9128
EC00954=34.0966,5355.0000
EC00955=34.1079,5358.0872
EC00956=33.9827,5361.0007
EC00957=31.6349,5363.6952
EC00958=19.5985,5365.3417
EC00959=7.5993,5366.3401
EC00960=2.6033,5367.0710
EC00961=1.0199,5367.7745
EC00962=0.7177,5368.7006
EC00963=0.1365,5370.2391
EC00964=-0.4862,5372.2062
EC00965=0.0128,5374.3302
EC00966=0.0000,5376.4460
EC00967=0.0000,5378.5542
EC00968=0.0181,5380.6701
EC00969=-0.4893,5382.7940
EC00970=0.1337,5384.7609
EC00971=0.7176,5386.2991
EC00972=1.0211,5387.2255
EC00973=2.6020,5387.9295
EC00974=7.5978,5388.6600
EC00975=19.6025,5389.6581
EC00976=31.6332,5391.3048
EC00977=33.9818,5393.9998
EC00978=34.1086,5396.9129
EC00979=34.0969,5400.0000
EC00980=34.1086,5403.0871
EC00981=33.9818,5406.0002
EC00982=31.6332,5408.6952
EC00983=19.6025,5410.3419
EC00984=7.5978,5411.3400
EC00985=2.6020,5412.0705
EC00986=1.0211,5412.7745
EC00987=0.7176,5413.7009
EC00988=0.1337,5415.2391
EC00989=-0.4893,5417.2060
EC00990=0.0181,5419.3299
EC00991=0.0000,5421.4458
EC00992=0.0000,5423.5540
EC00993=0.0128,5425.6698
EC00994=-0.4862,5427.7938
EC00995=0.1365,5429.7609
EC00996=0.7177,5431.2994
EC00997=1.0199,5432.2255
EC00998=2.6033,5432.9290
EC00999=7.5993,5433.6599
EC01000=19.5985,5434.6583
EC01001=31.6349,5436.3048
EC01002=33.9827,5438.9993
EC01003=34.1079,5441.9128
EC01004=34.0966,5445.0000
EC01005=34.1079,5448.0872
EC01006=33.9827,5451.0007
EC01007=31.6349,5453.6952
EC01008=19.5985,5455.3417
EC01009=7.5993,5456.3401
EC01010=2.6033,5457.0710
EC01011=1.0199,5457.7745
EC01012=0.7177,5458.7006
EC01013=0.1365,5460.2391
EC01014=-0.4862,5462.2062
EC01015=0.0128,5464.3302
EC01016=0.0000,5466.4460
EC01017=0.0000,5468.5542
EC01018=0.0181,5470.6701
EC01019=-0.4893,5472.7940
EC01020=0.1337,5474.7609
EC01021=0.7176,5476.2991
EC01022=1.0211,5477.2255
EC01023=2.6020,5477.9295
EC01024=7.5978,5478.6600
EC01025=19.6025,5479.6581
EC01026=31.6332,5481.3048
EC01027=33.9818,5483.9998
EC01028=34.1086,5486.9129
EC01029=34.0969,5490.0000
EC01030=35.0568,5490.0000
EC01031=35.0693,5493.0565
EC01032=34.9274,5495.9598
EC01033=32.1963,5498.6610
EC01034=17.9884,5500.2852
EC01035=6.0027,5501.2483
EC01036=1.6678,5501.9417
EC01037=0.2592,5502.6030
EC01038=-0.0575,5503.4837
EC01039=-0.2980,5505.0155
EC01040=-0.6721,5507.0162
EC01041=-0.0000,5509.2050
EC01042=-0.0000,5511.4028
EC01043=-0.0000,5513.5971
EC01044=-0.0000,5515.7952
EC01045=-0.6749,5517.9837
EC01046=-0.2926,5519.9842
EC01047=-0.0585,5521.5162
EC01048=0.2613,5522.3970
EC01049=1.6678,5523.0583
EC01050=6.0013,5523.7518
EC01051=17.9871,5524.7152
EC01052=32.1987,5526.3389
EC01053=34.9311,5529.0399
EC01054=35.0679,5531.9437
EC01055=35.0560,5535.0000
EC01056=35.0679,5538.0563
EC01057=34.9274,5540.9601
EC01058=32.1958,5543.6611
EC01059=17.9871,5545.2848
EC01060=6.0013,5546.2482
EC01061=1.6678,5546.9417
EC01062=0.2613,5547.6030
EC01063=-0.0585,5548.4838
EC01064=-0.2926,5550.0158
EC01065=-0.6749,5552.0163
EC01066=-0.0000,5554.2048
EC01067=-0.0000,5556.4029
EC01068=-0.0000,5558.5972
EC01069=-0.0000,5560.7950
EC01070=-0.6721,5562.9838
EC01071=-0.2980,5564.9845
EC01072=-0.0575,5566.5163
EC01073=0.2592,5567.3970
EC01074=1.6678,5568.0583
EC01075=6.0027,5568.7517
EC01076=17.9884,5569.7148
EC01077=32.1963,5571.3390
EC01078=34.9274,5574.0402
EC01079=35.0693,5576.9435
EC01080=35.0568,5580.0000
EC01081=35.0690,5583.0565
EC01082=34.9269,5585.9604
EC01083=32.1963,5588.6610
EC01084=17.9884,5590.2852
EC01085=6.0027,5591.2483
EC01086=1.6678,5591.9417
EC01087=0.2592,5592.6030
EC01088=-0.0575,5593.4837
EC01089=-0.2980,5595.0155
EC01090=-0.6721,5597.0162
EC01091=-0.0000,5599.2050
EC01092=-0.0000,5601.4028
EC01093=-0.0000,5603.5971
EC01094=-0.0000,5605.7952
EC01095=-0.6749,5607.9837
EC01096=-0.2926,5609.9842
EC01097=-0.0585,5611.5162
EC01098=0.2613,5612.3970
EC01099=1.6678,5613.0583
EC01100=6.0013,5613.7518
EC01101=17.9871,5614.7152
EC01102=32.1987,5616.3389
EC01103=34.9311,5619.0399
EC01104=35.0679,5621.9437
EC01105=35.0560,5625.0000
EC01106=35.0679,5628.0563
EC01107=34.9274,5630.9601
EC01108=32.1958,5633.6611
EC01109=17.9871,5635.2848
EC01110=6.0013,5636.2482
EC01111=1.6678,5636.9417
EC01112=0.2613,5637.6030
EC01113=-0.0585,5638.4838
EC01114=-0.2926,5640.0158
EC01115=-0.6749,5642.0163
EC01116=-0.0000,5644.2048
EC01117=-0.0000,5646.4029
EC01118=-0.0000,5648.5972
EC01119=-0.0000,5650.7950
EC01120=-0.6721,5652.9838
EC01121=-0.2980,5654.9845
EC01122=-0.0575,5656.5163
EC01123=0.2592,5657.3970
EC01124=1.6678,5658.0583
EC01125=6.0027,5658.7517
EC01126=17.9884,5659.7148
EC01127=32.1963,5661.3390
EC01128=34.9274,5664.0402
EC01129=35.0693,5666.9435
EC01130=35.0568,5670.0000
EC01131=35.0568,5670.0000
EC01132=35.0690,5673.0565
EC01133=34.9269,5675.9604
EC01134=32.1963,5678.6610
EC01135=17.9884,5680.2852
EC01136=6.0027,5681.2483
EC01137=1.6678,5681.9417
EC01138=0.2592,5682.6030
EC01139=-0.0575,5683.4837
EC01140=-0.2980,5685.0155
EC01141=-0.6721,5687.0162
EC01142=-0.0000,5689.2050
EC01143=-0.0000,5691.4028
EC01144=-0.0000,5693.5971
EC01145=-0.0000,5695.7952
EC01146=-0.6749,5697.9837
EC01147=-0.2926,5699.9842
EC01148=-0.0585,5701.5162
EC01149=0.2613,5702.3970
EC01150=1.6678,5703.0583
EC01151=6.0013,5703.7518
EC01152=17.9871,5704.7152
EC01153=32.1987,5706.3389
EC01154=34.9311,5709.0399
EC01155=35.0679,5711.9437
EC01156=35.0560,5715.0000
EC01157=35.0679,5718.0563
EC01158=34.9274,5720.9601
EC01159=32.1958,5723.6611
EC01160=17.9871,5725.2848
EC01161=6.0013,5726.2482
EC01162=1.6678,5726.9417
EC01163=0.2613,5727.6030
EC01164=-0.0585,5728.4838
EC01165=-0.2926,5730.0158
EC01166=-0.6749,5732.0163
EC01167=-0.0000,5734.2048
EC01168=-0.0000,5736.4029
EC01169=-0.0000,5738.5972
EC01170=-0.0000,5740.7950
EC01171=-0.6721,5742.9838
EC01172=-0.2980,5744.9845
EC01173=-0.0575,5746.5163
EC01174=0.2592,5747.3970
EC01175=1.6678,5748.0583
EC01176=6.0027,5748.7517
EC01177=17.9884,5749.7148
EC01178=32.1963,5751.3390
EC01179=34.9274,5754.0402
EC01180=35.0693,5756.9435
EC01181=35.0568,5760.0000
EC01182=35.0690,5763.0565
EC01183=34.9269,5765.9604
EC01184=32.1963,5768.6610
EC01185=17.9884,5770.2852
EC01186=6.0027,5771.2483
EC01187=1.6678,5771.9417
EC01188=0.2592,5772.6030
EC01189=-0.0575,5773.4837
EC01190=-0.2980,5775.0155
EC01191=-0.6721,5777.0162
EC01192=-0.0000,5779.2050
EC01193=-0.0000,5781.4028
EC01194=-0.0000,5783.5971
EC01195=-0.0000,5785.7952
EC01196=-0.6749,5787.9837
EC01197=-0.2926,5789.9842
EC01198=-0.0585,5791.5162
EC01199=0.2613,5792.3970
EC01200=1.6678,5793.0583
EC01201=6.0013,5793.7518
EC01202=17.9871,5794.7152
EC01203=32.1987,5796.3389
EC01204=34.9311,5799.0399
EC01205=35.0679,5801.9437
EC01206=35.0560,5805.0000
EC01207=35.0679,5808.0563
EC01208=34.9274,5810.9601
EC01209=32.1958,5813.6611
EC01210=17.9871,5815.2848
EC01211=6.0013,5816.2482
EC01212=1.6678,5816.9417
EC01213=0.2613,5817.6030
EC01214=-0.0585,5818.4838
EC01215=-0.2926,5820.0158
EC01216=-0.6749,5822.0163
EC01217=-0.0000,5824.2048
EC01218=-0.0000,5826.4029
EC01219=-0.0000,5828.5972
EC01220=-0.0000,5830.7950
EC01221=-0.6721,5832.9838
EC01222=-0.2980,5834.9845
EC01223=-0.0575,5836.5163
EC01224=0.2592,5837.3970
EC01225=1.6678,5838.0583
EC01226=6.0027,5838.7517
EC01227=17.9884,5839.7148
EC01228=32.1963,5841.3390
EC01229=34.9269,5844.0396
EC01230=35.0690,5846.9435
EC01231=35.0568,5850.0000
EC01232=35.8947,5850.0000
EC01233=35.9073,5853.0242
EC01234=35.7506,5855.9175
EC01235=32.5775,5858.6252
EC01236=16.1560,5860.2250
EC01237=4.6136,5861.1519
EC01238=0.9554,5861.8065
EC01239=-0.3032,5862.4248
EC01240=-0.7502,5863.2580
EC01241=-0.7251,5864.7847
EC01242=-0.8662,5866.8204
EC01243=-0.0181,5869.0758
EC01244=-0.0053,5871.3580
EC01245=-0.0052,5873.6417
EC01246=-0.0180,5875.9241
EC01247=-0.8665,5878.1796
EC01248=-0.7285,5880.2155
EC01249=-0.7508,5881.7418
EC01250=-0.3053,5882.5751
EC01251=0.9541,5883.1936
EC01252=4.6171,5883.8475
EC01253=16.1553,5884.7753
EC01254=32.5797,5886.3747
EC01255=35.7490,5889.0826
EC01256=35.9085,5891.9754
EC01257=35.8962,5895.0000
EC01258=35.9085,5898.0237
EC01259=35.7490,5900.9174
EC01260=32.5797,5903.6253
EC01261=16.1553,5905.2247
EC01262=4.6171,5906.1525
EC01263=0.9541,5906.8064
EC01264=-0.3053,5907.4249
EC01265=-0.7508,5908.2582
EC01266=-0.7285,5909.7845
EC01267=-0.8665,5911.8204
EC01268=-0.0180,5914.0759
EC01269=-0.0052,5916.3583
EC01270=-0.0053,5918.6420
EC01271=-0.0181,5920.9242
EC01272=-0.8662,5923.1796
EC01273=-0.7251,5925.2153
EC01274=-0.7502,5926.7420
EC01275=-0.3032,5927.5752
EC01276=0.9554,5928.1935
EC01277=4.6136,5928.8481
EC01278=16.1560,5929.7750
EC01279=32.5775,5931.3748
EC01280=35.7506,5934.0825
EC01281=35.9073,5936.9758
EC01282=35.8947,5940.0000
EC01283=35.9073,5943.0242
EC01284=35.7506,5945.9175
EC01285=32.5775,5948.6252
EC01286=16.1560,5950.2250
EC01287=4.6136,5951.1519
EC01288=0.9554,5951.8065
EC01289=-0.3032,5952.4248
EC01290=-0.7502,5953.2580
EC01291=-0.7251,5954.7847
EC01292=-0.8662,5956.8204
EC01293=-0.0181,5959.0758
EC01294=-0.0053,5961.3580
EC01295=-0.0052,5963.6417
EC01296=-0.0180,5965.9241
EC01297=-0.8665,5968.1796
EC01298=-0.7285,5970.2155
EC01299=-0.7508,5971.7418
EC01300=-0.3053,5972.5751
EC01301=0.9541,5973.1936
EC01302=4.6171,5973.8475
EC01303=16.1553,5974.7753
EC01304=32.5797,5976.3747
EC01305=35.7490,5979.0826
EC01306=35.9085,5981.9754
EC01307=35.8962,5985.0000
EC01308=35.9085,5988.0237
EC01309=35.7490,5990.9174
EC01310=32.5797,5993.6253
EC01311=16.1553,5995.2247
EC01312=4.6171,5996.1525
EC01313=0.9541,5996.8064
EC01314=-0.3053,5997.4249
EC01315=-0.7508,5998.2582
EC01316=-0.7285,5999.7845
EC01317=-0.8665,6001.8204
EC01318=-0.0180,6004.0759
EC01319=-0.0052,6006.3583
EC01320=-0.0053,6008.6420
EC01321=-0.0181,6010.9242
EC01322=-0.8662,6013.1796
EC01323=-0.7251,6015.2153
EC01324=-0.7502,6016.7420
EC01325=-0.3032,6017.5752
EC01326=0.9554,6018.1935
EC01327=4.6136,6018.8481
EC01328=16.1560,6019.7750
EC01329=32.5775,6021.3748
EC01330=35.7506,6024.0825
EC01331=35.9073,6026.9758
EC01332=35.8947,6030.0000
EC01333=35.8947,6030.0000
EC01334=35.9073,6033.0242
EC01335=35.7506,6035.9175
EC01336=32.5775,6038.6252
EC01337=16.1560,6040.2250
EC01338=4.6136,6041.1519
EC01339=0.9554,6041.8065
EC01340=-0.3032,6042.4248
EC01341=-0.7502,6043.2580
EC01342=-0.7251,6044.7847
EC01343=-0.8662,6046.8204
EC01344=-0.0181,6049.0758
EC01345=-0.0053,6051.3580
EC01346=-0.0052,6053.6417
EC01347=-0.0180,6055.9241
EC01348=-0.8665,6058.1796
EC01349=-0.7285,6060.2155
EC01350=-0.7508,6061.7418
EC01351=-0.3053,6062.5751
EC01352=0.9541,6063.1936
EC01353=4.6171,6063.8475
EC01354=16.1553,6064.7753
EC01355=32.5797,6066.3747
EC01356=35.7490,6069.0826
EC01357=35.9085,6071.9754
EC01358=35.8962,6075.0000
EC01359=35.9085,6078.0237
EC01360=35.7490,6080.9174
EC01361=32.5797,6083.6253
EC01362=16.1553,6085.2247
EC01363=4.6171,6086.1525
EC01364=0.9541,6086.8064
EC01365=-0.3053,6087.4249
EC01366=-0.7508,6088.2582
EC01367=-0.7285,6089.7845
EC01368=-0.8665,6091.8204
EC01369=-0.0180,6094.0759
EC01370=-0.0052,6096.3583
EC01371=-0.0053,6098.6420
EC01372=-0.0181,6100.9242
EC01373=-0.8662,6103.1796
EC01374=-0.7251,6105.2153
EC01375=-0.7502,6106.7420
EC01376=-0.3032,6107.5752
EC01377=0.9554,6108.1935
EC01378=4.6136,6108.8481
EC01379=16.1560,6109.7750
EC01380=32.5775,6111.3748
EC01381=35.7506,6114.0825
EC01382=35.9073,6116.9758
EC01383=35.8947,6120.0000
EC01384=35.9073,6123.0242
EC01385=35.7506,6125.9175
EC01386=32.5775,6128.6252
EC01387=16.1560,6130.2250
EC01388=4.6136,6131.1519
EC01389=0.9554,6131.8065
EC01390=-0.3032,6132.4248
EC01391=-0.7502,6133.2580
EC01392=-0.7251,6134.7847
EC01393=-0.8662,6136.8204
EC01394=-0.0181,6139.0758
EC01395=-0.0053,6141.3580
EC01396=-0.0052,6143.6417
EC01397=-0.0180,6145.9241
EC01398=-0.8665,6148.1796
EC01399=-0.7285,6150.2155
EC01400=-0.7508,6151.7418
EC01401=-0.3053,6152.5751
EC01402=0.9541,6153.1936
EC01403=4.6171,6153.8475
EC01404=16.1553,6154.7753
EC01405=32.5797,6156.3747
EC01406=35.7490,6159.0826
EC01407=35.9085,6161.9754
EC01408=35.8962,6165.0000
EC01409=35.9085,6168.0237
EC01410=35.7490,6170.9174
EC01411=32.5797,6173.6253
EC01412=16.1553,6175.2247
EC01413=4.6171,6176.1525
EC01414=0.9541,6176.8064
EC01415=-0.3053,6177.4249
EC01416=-0.7508,6178.2582
EC01417=-0.7285,6179.7845
EC01418=-0.8665,6181.8204
EC01419=-0.0180,6184.0759
EC01420=-0.0052,6186.3583
EC01421=-0.0053,6188.6420
EC01422=-0.0181,6190.9242
EC01423=-0.8662,6193.1796
EC01424=-0.7251,6195.2153
EC01425=-0.7502,6196.7420
EC01426=-0.3032,6197.5752
EC01427=0.9554,6198.1935
EC01428=4.6136,6198.8481
EC01429=16.1560,6199.7750
EC01430=32.5775,6201.3748
EC01431=35.7506,6204.0825
EC01432=35.9073,6206.9758
EC01433=35.8947,6210.0000
EC01434=36.6281,6210.0000
EC01435=36.6409,6212.9903
EC01436=36.4598,6215.8729
EC01437=32.7893,6218.5881
EC01438=14.2031,6220.1621
EC01439=3.4506,6221.0515
EC01440=0.4238,6221.6656
EC01441=-0.7002,6222.2395
EC01442=-1.3423,6223.0258
EC01443=-1.1510,6224.5467
EC01444=-1.0519,6226.6187
EC01445=-0.0362,6228.9437
EC01446=-0.0053,6231.3119
EC01447=-0.0052,6233.6874
EC01448=-0.0333,6236.0569
EC01449=-1.0536,6238.3812
EC01450=-1.1484,6240.4534
EC01451=-1.3439,6241.9748
EC01452=-0.6999,6242.7607
EC01453=0.4261,6243.3343
EC01454=3.4541,6243.9482
EC01455=14.2058,6244.8381
EC01456=32.7883,6246.4120
EC01457=36.4603,6249.1268
EC01458=36.6399,6252.0095
EC01459=36.6307,6255.0000
EC01460=36.6399,6257.9905
EC01461=36.4603,6260.8732
EC01462=32.7883,6263.5880
EC01463=14.2058,6265.1619
EC01464=3.4541,6266.0518
EC01465=0.4261,6266.6657
EC01466=-0.6999,6267.2393
EC01467=-1.3439,6268.0252
EC01468=-1.1484,6269.5466
EC01469=-1.0536,6271.6188
EC01470=-0.0333,6273.9431
EC01471=-0.0052,6276.3126
EC01472=-0.0053,6278.6881
EC01473=-0.0362,6281.0563
EC01474=-1.0519,6283.3813
EC01475=-1.1510,6285.4533
EC01476=-1.3423,6286.9742
EC01477=-0.7002,6287.7605
EC01478=0.4238,6288.3344
EC01479=3.4506,6288.9485
EC01480=14.2031,6289.8379
EC01481=32.7893,6291.4119
EC01482=36.4598,6294.1271
EC01483=36.6409,6297.0097
EC01484=36.6281,6300.0000
EC01485=36.6409,6302.9903
EC01486=36.4598,6305.8729
EC01487=32.7900,6308.5881
EC01488=14.2031,6310.1621
EC01489=3.4506,6311.0515
EC01490=0.4238,6311.6656
EC01491=-0.7002,6312.2395
EC01492=-1.3423,6313.0258
EC01493=-1.1510,6314.5467
EC01494=-1.0519,6316.6187
EC01495=-0.0362,6318.9437
EC01496=-0.0053,6321.3119
EC01497=-0.0052,6323.6874
EC01498=-0.0333,6326.0569
EC01499=-1.0536,6328.3812
EC01500=-1.1484,6330.4534
EC01501=-1.3439,6331.9748
EC01502=-0.6999,6332.7607
EC01503=0.4261,6333.3343
EC01504=3.4541,6333.9482
EC01505=14.2058,6334.8381
EC01506=32.7883,6336.4120
EC01507=36.4603,6339.1268
EC01508=36.6399,6342.0095
EC01509=36.6307,6345.0000
EC01510=36.6399,6347.9905
EC01511=36.4603,6350.8732
EC01512=32.7883,6353.5880
EC01513=14.2058,6355.1619
EC01514=3.4541,6356.0518
EC01515=0.4261,6356.6657
EC01516=-0.6999,6357.2393
EC01517=-1.3439,6358.0252
EC01518=-1.1484,6359.5466
EC01519=-1.0536,6361.6188
EC01520=-0.0333,6363.9431
EC01521=-0.0052,6366.3126
EC01522=-0.0053,6368.6881
EC01523=-0.0362,6371.0563
EC01524=-1.0519,6373.3813
EC01525=-1.1510,6375.4533
EC01526=-1.3423,6376.9742
EC01527=-0.7002,6377.7605
EC01528=0.4238,6378.3344
EC01529=3.4506,6378.9485
EC01530=14.2031,6379.8379
EC01531=32.7893,6381.4119
EC01532=36.4598,6384.1271
EC01533=36.6409,6387.0097
EC01534=36.6281,6390.0000
EC01535=36.6281,6390.0000
EC01536=36.6409,6392.9903
EC01537=36.4598,6395.8729
EC01538=32.7900,6398.5881
EC01539=14.2031,6400.1621
EC01540=3.4506,6401.0515
EC01541=0.4238,6401.6656
EC01542=-0.7002,6402.2395
EC01543=-1.3423,6403.0258
EC01544=-1.1510,6404.5467
EC01545=-1.0519,6406.6187
EC01546=-0.0362,6408.9437
EC01547=-0.0053,6411.3119
EC01548=-0.0052,6413.6874
EC01549=-0.0333,6416.0569
EC01550=-1.0536,6418.3812
EC01551=-1.1484,6420.4534
EC01552=-1.3439,6421.9748
EC01553=-0.6999,6422.7607
EC01554=0.4261,6423.3343
EC01555=3.4541,6423.9482
EC01556=14.2058,6424.8381
EC01557=32.7883,6426.4120
EC01558=36.4603,6429.1268
EC01559=36.6399,6432.0095
EC01560=36.6307,6435.0000
EC01561=36.6399,6437.9905
EC01562=36.4603,6440.8732
EC01563=32.7883,6443.5880
EC01564=14.2058,6445.1619
EC01565=3.4541,6446.0518
EC01566=0.4261,6446.6657
EC01567=-0.6999,6447.2393
EC01568=-1.3439,6448.0252
EC01569=-1.1484,6449.5466
EC01570=-1.0536,6451.6188
EC01571=-0.0333,6453.9431
EC01572=-0.0052,6456.3126
EC01573=-0.0053,6458.6881
EC01574=-0.0362,6461.0563
EC01575=-1.0519,6463.3813
EC01576=-1.1510,6465.4533
EC01577=-1.3423,6466.9742
EC01578=-0.7002,6467.7605
EC01579=0.4238,6468.3344
EC01580=3.4506,6468.9485
EC01581=14.2031,6469.8379
EC01582=32.7893,6471.4119
EC01583=36.4598,6474.1271
EC01584=36.6409,6477.0097
EC01585=36.6281,6480.0000
EC01586=36.6409,6482.9903
EC01587=36.4598,6485.8729
EC01588=32.7900,6488.5881
EC01589=14.2031,6490.1621
EC01590=3.4506,6491.0515
EC01591=0.4238,6491.6656
EC01592=-0.7002,6492.2395
EC01593=-1.3423,6493.0258
EC01594=-1.1510,6494.5467
EC01595=-1.0519,6496.6187
EC01596=-0.0362,6498.9437
EC01597=-0.0053,6501.3119
EC01598=-0.0052,6503.6874
EC01599=-0.0333,6506.0569
EC01600=-1.0536,6508.3812
EC01601=-1.1484,6510.4534
EC01602=-1.3439,6511.9748
EC01603=-0.6999,6512.7607
EC01604=0.4261,6513.3343
EC01605=3.4541,6513.9482
EC01606=14.2058,6514.8381
EC01607=32.7883,6516.4120
EC01608=36.4603,6519.1268
EC01609=36.6399,6522.0095
EC01610=36.6307,6525.0000
EC01611=36.6399,6527.9905
EC01612=36.4603,6530.8732
EC01613=32.7883,6533.5880
EC01614=14.2058,6535.1619
EC01615=3.4541,6536.0518
EC01616=0.4261,6536.6657
EC01617=-0.6999,6537.2393
EC01618=-1.3439,6538.0252
EC01619=-1.1484,6539.5466
EC01620=-1.0536,6541.6188
EC01621=-0.0333,6543.9431
EC01622=-0.0052,6546.3126
EC01623=-0.0053,6548.6881
EC01624=-0.0362,6551.0563
EC01625=-1.0519,6553.3813
EC01626=-1.1510,6555.4533
EC01627=-1.3423,6556.9742
EC01628=-0.7002,6557.7605
EC01629=0.4238,6558.3344
EC01630=3.4506,6558.9485
EC01631=14.2031,6559.8379
EC01632=32.7900,6561.4119
EC01633=36.4598,6564.1271
EC01634=36.6409,6567.0097
EC01635=36.6281,6570.0000
EC01636=37.2584,6570.0000
EC01637=37.2713,6572.9548
EC01638=37.0692,6575.8263
EC01639=32.8316,6578.5486
EC01640=12.2420,6580.0964
EC01641=2.5084,6580.9471
EC01642=0.0477,6581.5198
EC01643=-0.9486,6582.0484
EC01644=-1.8150,6582.7860
EC01645=-1.5540,6584.3034
EC01646=-1.2364,6586.4132
EC01647=-0.0489,6588.8079
EC01648=-0.0053,6591.2653
EC01649=-0.0076,6593.7346
EC01650=-0.0512,6596.1917
EC01651=-1.2364,6598.5867
EC01652=-1.5518,6600.6966
EC01653=-1.8116,6602.2136
EC01654=-0.9491,6602.9519
EC01655=0.0487,6603.4806
EC01656=2.5069,6604.0527
EC01657=12.2381,6604.9034
EC01658=32.8330,6606.4513
EC01659=37.0682,6609.1737
EC01660=37.2688,6612.0450
EC01661=37.2595,6615.0000
EC01662=37.2688,6617.9550
EC01663=37.0682,6620.8263
EC01664=32.8330,6623.5487
EC01665=12.2381,6625.0966
EC01666=2.5069,6625.9473
EC01667=0.0487,6626.5194
EC01668=-0.9491,6627.0481
EC01669=-1.8116,6627.7864
EC01670=-1.5518,6629.3034
EC01671=-1.2364,6631.4133
EC01672=-0.0512,6633.8083
EC01673=-0.0076,6636.2654
EC01674=-0.0053,6638.7347
EC01675=-0.0489,6641.1921
EC01676=-1.2364,6643.5868
EC01677=-1.5540,6645.6966
EC01678=-1.8150,6647.2140
EC01679=-0.9486,6647.9516
EC01680=0.0477,6648.4802
EC01681=2.5084,6649.0529
EC01682=12.2420,6649.9036
EC01683=32.8316,6651.4514
EC01684=37.0692,6654.1737
EC01685=37.2713,6657.0452
EC01686=37.2584,6660.0000
EC01687=37.2713,6662.9548
EC01688=37.0687,6665.8263
EC01689=32.8316,6668.5486
EC01690=12.2420,6670.0964
EC01691=2.5084,6670.9471
EC01692=0.0477,6671.5198
EC01693=-0.9486,6672.0484
EC01694=-1.8150,6672.7860
EC01695=-1.5540,6674.3034
EC01696=-1.2364,6676.4132
EC01697=-0.0489,6678.8079
EC01698=-0.0053,6681.2653
EC01699=-0.0076,6683.7346
EC01700=-0.0512,6686.1917
EC01701=-1.2364,6688.5867
EC01702=-1.5518,6690.6966
EC01703=-1.8116,6692.2136
EC01704=-0.9491,6692.9519
EC01705=0.0487,6693.4806
EC01706=2.5069,6694.0527
EC01707=12.2381,6694.9034
EC01708=32.8330,6696.4513
EC01709=37.0682,6699.1737
EC01710=37.2688,6702.0450
EC01711=37.2595,6705.0000
EC01712=37.2688,6707.9550
EC01713=37.0682,6710.8263
EC01714=32.8330,6713.5487
EC01715=12.2381,6715.0966
EC01716=2.5069,6715.9473
EC01717=0.0487,6716.5194
EC01718=-0.9491,6717.0481
EC01719=-1.8116,6717.7864
EC01720=-1.5518,6719.3034
EC01721=-1.2364,6721.4133
EC01722=-0.0512,6723.8083
EC01723=-0.0076,6726.2654
EC01724=-0.0053,6728.7347
EC01725=-0.0489,6731.1921
EC01726=-1.2364,6733.5868
EC01727=-1.5540,6735.6966
EC01728=-1.8150,6737.2140
EC01729=-0.9486,6737.9516
EC01730=0.0477,6738.4802
EC01731=2.5084,6739.0529
EC01732=12.2420,6739.9036
EC01733=32.8316,6741.4514
EC01734=37.0692,6744.1737
EC01735=37.2713,6747.0452
EC01736=37.2584,6750.0000
EC01737=37.2584,6750.0000
EC01738=37.2713,6752.9548
EC01739=37.0687,6755.8263
EC01740=32.8316,6758.5486
EC01741=12.2420,6760.0964
EC01742=2.5084,6760.9471
EC01743=0.0477,6761.5198
EC01744=-0.9486,6762.0484
EC01745=-1.8150,6762.7860
EC01746=-1.5540,6764.3034
EC01747=-1.2364,6766.4132
EC01748=-0.0489,6768.8079
EC01749=-0.0053,6771.2653
EC01750=-0.0076,6773.7346
EC01751=-0.0512,6776.1917
EC01752=-1.2364,6778.5867
EC01753=-1.5518,6780.6966
EC01754=-1.8116,6782.2136
EC01755=-0.9491,6782.9519
EC01756=0.0487,6783.4806
EC01757=2.5069,6784.0527
EC01758=12.2381,6784.9034
EC01759=32.8330,6786.4513
EC01760=37.0682,6789.1737
EC01761=37.2688,6792.0450
EC01762=37.2595,6795.0000
EC01763=37.2688,6797.9550
EC01764=37.0682,6800.8263
EC01765=32.8330,6803.5487
EC01766=12.2381,6805.0966
EC01767=2.5069,6805.9473
EC01768=0.0487,6806.5194
EC01769=-0.9491,6807.0481
EC01770=-1.8116,6807.7864
EC01771=-1.5518,6809.3034
EC01772=-1.2364,6811.4133
EC01773=-0.0512,6813.8083
EC01774=-0.0076,6816.2654
EC01775=-0.0053,6818.7347
EC01776=-0.0489,6821.1921
EC01777=-1.2364,6823.5868
EC01778=-1.5540,6825.6966
EC01779=-1.8150,6827.2140
EC01780=-0.9486,6827.9516
EC01781=0.0477,6828.4802
EC01782=2.5084,6829.0529
EC01783=12.2420,6829.9036
EC01784=32.8316,6831.4514
EC01785=37.0692,6834.1737
EC01786=37.2713,6837.0452
EC01787=37.2584,6840.0000
EC01788=37.2713,6842.9548
EC01789=37.0687,6845.8263
EC01790=32.8316,6848.5486
EC01791=12.2420,6850.0964
EC01792=2.5084,6850.9471
EC01793=0.0477,6851.5198
EC01794=-0.9486,6852.0484
EC01795=-1.8150,6852.7860
EC01796=-1.5540,6854.3034
EC01797=-1.2364,6856.4132
EC01798=-0.0489,6858.8079
EC01799=-0.0053,6861.2653
EC01800=-0.0076,6863.7346
EC01801=-0.0512,6866.1917
EC01802=-1.2364,6868.5867
EC01803=-1.5518,6870.6966
EC01804=-1.8116,6872.2136
EC01805=-0.9491,6872.9519
EC01806=0.0487,6873.4806
EC01807=2.5069,6874.0527
EC01808=12.2381,6874.9034
EC01809=32.8330,6876.4513
EC01810=37.0682,6879.1737
EC01811=37.2688,6882.0450
EC01812=37.2595,6885.0000
EC01813=37.2688,6887.9550
EC01814=37.0682,6890.8263
EC01815=32.8330,6893.5487
EC01816=12.2381,6895.0966
EC01817=2.5069,6895.9473
EC01818=0.0487,6896.5194
EC01819=-0.9491,6897.0481
EC01820=-1.8116,6897.7864
EC01821=-1.5518,6899.3034
EC01822=-1.2364,6901.4133
EC01823=-0.0512,6903.8083
EC01824=-0.0076,6906.2654
EC01825=-0.0053,6908.7347
EC01826=-0.0489,6911.1921
EC01827=-1.2364,6913.5868
EC01828=-1.5540,6915.6966
EC01829=-1.8150,6917.2140
EC01830=-0.9486,6917.9516
EC01831=0.0477,6918.4802
EC01832=2.5084,6919.0529
EC01833=12.2420,6919.9036
EC01834=32.8316,6921.4514
EC01835=37.0687,6924.1737
EC01836=37.2713,6927.0452
EC01837=37.2584,6930.0000
EC01838=37.7936,6930.0000
EC01839=37.8064,6932.9180
EC01840=37.5779,6935.7775
EC01841=32.7139,6938.5076
EC01842=10.3506,6940.0280
EC01843=1.7602,6940.8382
EC01844=-0.2048,6941.3683
EC01845=-1.0819,6941.8512
EC01846=-2.1680,6942.5410
EC01847=-1.9251,6944.0550
EC01848=-1.4088,6946.2037
EC01849=-0.0652,6948.6701
EC01850=-0.0074,6951.2180
EC01851=-0.0076,6953.7821
EC01852=-0.0641,6956.3297
EC01853=-1.4120,6958.7961
EC01854=-1.9264,6960.9450
EC01855=-2.1668,6962.4587
EC01856=-1.0827,6963.1487
EC01857=-0.2057,6963.6320
EC01858=1.7614,6964.1614
EC01859=10.3507,6964.9722
EC01860=32.7126,6966.4919
EC01861=37.5797,6969.2230
EC01862=37.8051,6972.0820
EC01863=37.7926,6975.0000
EC01864=37.8051,6977.9180
EC01865=37.5797,6980.7770
EC01866=32.7166,6983.5081
EC01867=10.3507,6985.0278
EC01868=1.7614,6985.8386
EC01869=-0.2057,6986.3680
EC01870=-1.0827,6986.8513
EC01871=-2.1668,6987.5413
EC01872=-1.9264,6989.0550
EC01873=-1.4120,6991.2039
EC01874=-0.0641,6993.6703
EC01875=-0.0076,6996.2179
EC01876=-0.0074,6998.7820
EC01877=-0.0652,7001.3299
EC01878=-1.4088,7003.7963
EC01879=-1.9251,7005.9450
EC01880=-2.1680,7007.4590
EC01881=-1.0819,7008.1488
EC01882=-0.2048,7008.6317
EC01883=1.7602,7009.1618
EC01884=10.3506,7009.9720
EC01885=32.7139,7011.4924
EC01886=37.5779,7014.2225
EC01887=37.8064,7017.0820
EC01888=37.7936,7020.0000
EC01889=37.8064,7022.9180
EC01890=37.5779,7025.7775
EC01891=32.7146,7028.5076
EC01892=10.3506,7030.0280
EC01893=1.7602,7030.8382
EC01894=-0.2048,7031.3683
EC01895=-1.0819,7031.8512
EC01896=-2.1680,7032.5410
EC01897=-1.9251,7034.0550
EC01898=-1.4088,7036.2037
EC01899=-0.0652,7038.6701
EC01900=-0.0074,7041.2180
EC01901=-0.0076,7043.7821
EC01902=-0.0641,7046.3297
EC01903=-1.4120,7048.7961
EC01904=-1.9264,7050.9450
EC01905=-2.1668,7052.4587
EC01906=-1.0827,7053.1487
EC01907=-0.2057,7053.6320
EC01908=1.7614,7054.1614
EC01909=10.3507,7054.9722
EC01910=32.7126,7056.4919
EC01911=37.5797,7059.2230
EC01912=37.8051,7062.0820
EC01913=37.7926,7065.0000
EC01914=37.8051,7067.9180
EC01915=37.5797,7070.7770
EC01916=32.7166,7073.5081
EC01917=10.3507,7075.0278
EC01918=1.7614,7075.8386
EC01919=-0.2057,7076.3680
EC01920=-1.0827,7076.8513
EC01921=-2.1668,7077.5413
EC01922=-1.9264,7079.0550
EC01923=-1.4120,7081.2039
EC01924=-0.0641,7083.6703
EC01925=-0.0076,7086.2179
EC01926=-0.0074,7088.7820
EC01927=-0.0652,7091.3299
EC01928=-1.4088,7093.7963
EC01929=-1.9251,7095.9450
EC01930=-2.1680,7097.4590
EC01931=-1.0819,7098.1488
EC01932=-0.2048,7098.6317
EC01933=1.7602,7099.1618
EC01934=10.3506,7099.9720
EC01935=32.7139,7101.4924
EC01936=37.5779,7104.2225
EC01937=37.8064,7107.0820
EC01938=37.7936,7110.0000
EC01939=37.7936,7110.0000
EC01940=37.8064,7112.9180
EC01941=37.5779,7115.7775
EC01942=32.7146,7118.5076
EC01943=10.3506,7120.0280
EC01944=1.7602,7120.8382
EC01945=-0.2048,7121.3683
EC01946=-1.0819,7121.8512
EC01947=-2.1680,7122.5410
EC01948=-1.9251,7124.0550
EC01949=-1.4088,7126.2037
EC01950=-0.0652,7128.6701
EC01951=-0.0074,7131.2180
EC01952=-0.0076,7133.7821
EC01953=-0.0641,7136.3297
EC01954=-1.4120,7138.7961
EC01955=-1.9264,7140.9450
EC01956=-2.1668,7142.4587
EC01957=-1.0827,7143.1487
EC01958=-0.2057,7143.6320
EC01959=1.7614,7144.1614
EC01960=10.3507,7144.9722
EC01961=32.7126,7146.4919
EC01962=37.5797,7149.2230
EC01963=37.8051,7152.0820
EC01964=37.7926,7155.0000
EC01965=37.8051,7157.9180
EC01966=37.5797,7160.7770
EC01967=32.7166,7163.5081
EC01968=10.3507,7165.0278
EC01969=1.7614,7165.8386
EC01970=-0.2057,7166.3680
EC01971=-1.0827,7166.8513
EC01972=-2.1668,7167.5413
EC01973=-1.9264,7169.0550
EC01974=-1.4120,7171.2039
EC01975=-0.0641,7173.6703
EC01976=-0.0076,7176.2179
EC01977=-0.0074,7178.7820
EC01978=-0.0652,7181.3299
EC01979=-1.4088,7183.7963
EC01980=-1.9251,7185.9450
EC01981=-2.1680,7187.4590
EC01982=-1.0819,7188.1488
EC01983=-0.2048,7188.6317
EC01984=1.7602,7189.1618
EC01985=10.3506,7189.9720
EC01986=32.7139,7191.4924
EC01987=37.5779,7194.2225
EC01988=37.8064,7197.0820
EC01989=37.7936,7200.0000
EC01990=37.8064,7202.9180
EC01991=37.5779,7205.7775
EC01992=32.7146,7208.5076
EC01993=10.3506,7210.0280
EC01994=1.7602,7210.8382
EC01995=-0.2048,7211.3683
EC01996=-1.0819,7211.8512
EC01997=-2.1680,7212.5410
EC01998=-1.9251,7214.0550
EC01999=-1.4088,7216.2037
//INST
///DATE 2021/09/24 14:36
///COMM
///ATTR SC,RW,RJ
////FRAME USER 2
///GROUP1 RB1
///GROUP2 ST1
NOP
SMOVL C00000 +MOVJ EC00000
SMOVL C00001 +MOVJ EC00001
SMOVL C00002 +MOVJ EC00002
SMOVL C00003 +MOVJ EC00003
SMOVL C00004 +MOVJ EC00004
SMOVL C00005 +MOVJ EC00005
SMOVL C00006 +MOVJ EC00006
SMOVL C00007 +MOVJ EC00007
SMOVL C00008 +MOVJ EC00008
SMOVL C00009 +MOVJ EC00009
SMOVL C00010 +MOVJ EC00010
SMOVL C00011 +MOVJ EC00011
SMOVL C00012 +MOVJ EC00012
SMOVL C00013 +MOVJ EC00013
SMOVL C00014 +MOVJ EC00014
SMOVL C00015 +MOVJ EC00015
SMOVL C00016 +MOVJ EC00016
SMOVL C00017 +MOVJ EC00017
SMOVL C00018 +MOVJ EC00018
SMOVL C00019 +MOVJ EC00019
SMOVL C00020 +MOVJ EC00020
SMOVL C00021 +MOVJ EC00021
SMOVL C00022 +MOVJ EC00022
SMOVL C00023 +MOVJ EC00023
SMOVL C00024 +MOVJ EC00024
SMOVL C00025 +MOVJ EC00025
SMOVL C00026 +MOVJ EC00026
SMOVL C00027 +MOVJ EC00027
SMOVL C00028 +MOVJ EC00028
SMOVL C00029 +MOVJ EC00029
SMOVL C00030 +MOVJ EC00030
SMOVL C00031 +MOVJ EC00031
SMOVL C00032 +MOVJ EC00032
SMOVL C00033 +MOVJ EC00033
SMOVL C00034 +MOVJ EC00034
SMOVL C00035 +MOVJ EC00035
SMOVL C00036 +MOVJ EC00036
SMOVL C00037 +MOVJ EC00037
SMOVL C00038 +MOVJ EC00038
SMOVL C00039 +MOVJ EC00039
SMOVL C00040 +MOVJ EC00040
SMOVL C00041 +MOVJ EC00041
SMOVL C00042 +MOVJ EC00042
SMOVL C00043 +MOVJ EC00043
SMOVL C00044 +MOVJ EC00044
SMOVL C00045 +MOVJ EC00045
SMOVL C00046 +MOVJ EC00046
SMOVL C00047 +MOVJ EC00047
SMOVL C00048 +MOVJ EC00048
SMOVL C00049 +MOVJ EC00049
SMOVL C00050 +MOVJ EC00050
SMOVL C00051 +MOVJ EC00051
SMOVL C00052 +MOVJ EC00052
SMOVL C00053 +MOVJ EC00053
SMOVL C00054 +MOVJ EC00054
SMOVL C00055 +MOVJ EC00055
SMOVL C00056 +MOVJ EC00056
SMOVL C00057 +MOVJ EC00057
SMOVL C00058 +MOVJ EC00058
SMOVL C00059 +MOVJ EC00059
SMOVL C00060 +MOVJ EC00060
SMOVL C00061 +MOVJ EC00061
SMOVL C00062 +MOVJ EC00062
SMOVL C00063 +MOVJ EC00063
SMOVL C00064 +MOVJ EC00064
SMOVL C00065 +MOVJ EC00065
SMOVL C00066 +MOVJ EC00066
SMOVL C00067 +MOVJ EC00067
SMOVL C00068 +MOVJ EC00068
SMOVL C00069 +MOVJ EC00069
SMOVL C00070 +MOVJ EC00070
SMOVL C00071 +MOVJ EC00071
SMOVL C00072 +MOVJ EC00072
SMOVL C00073 +MOVJ EC00073
SMOVL C00074 +MOVJ EC00074
SMOVL C00075 +MOVJ EC00075
SMOVL C00076 +MOVJ EC00076
SMOVL C00077 +MOVJ EC00077
SMOVL C00078 +MOVJ EC00078
SMOVL C00079 +MOVJ EC00079
SMOVL C00080 +MOVJ EC00080
SMOVL C00081 +MOVJ EC00081
SMOVL C00082 +MOVJ EC00082
SMOVL C00083 +MOVJ EC00083
SMOVL C00084 +MOVJ EC00084
SMOVL C00085 +MOVJ EC00085
SMOVL C00086 +MOVJ EC00086
SMOVL C00087 +MOVJ EC00087
SMOVL C00088 +MOVJ EC00088
SMOVL C00089 +MOVJ EC00089
SMOVL C00090 +MOVJ EC00090
SMOVL C00091 +MOVJ EC00091
SMOVL C00092 +MOVJ EC00092
SMOVL C00093 +MOVJ EC00093
SMOVL C00094 +MOVJ EC00094
SMOVL C00095 +MOVJ EC00095
SMOVL C00096 +MOVJ EC00096
SMOVL C00097 +MOVJ EC00097
SMOVL C00098 +MOVJ EC00098
SMOVL C00099 +MOVJ EC00099
SMOVL C00100 +MOVJ EC00100
SMOVL C00101 +MOVJ EC00101
SMOVL C00102 +MOVJ EC00102
SMOVL C00103 +MOVJ EC00103
SMOVL C00104 +MOVJ EC00104
SMOVL C00105 +MOVJ EC00105
SMOVL C00106 +MOVJ EC00106
SMOVL C00107 +MOVJ EC00107
SMOVL C00108 +MOVJ EC00108
SMOVL C00109 +MOVJ EC00109
SMOVL C00110 +MOVJ EC00110
SMOVL C00111 +MOVJ EC00111
SMOVL C00112 +MOVJ EC00112
SMOVL C00113 +MOVJ EC00113
SMOVL C00114 +MOVJ EC00114
SMOVL C00115 +MOVJ EC00115
SMOVL C00116 +MOVJ EC00116
SMOVL C00117 +MOVJ EC00117
SMOVL C00118 +MOVJ EC00118
SMOVL C00119 +MOVJ EC00119
SMOVL C00120 +MOVJ EC00120
SMOVL C00121 +MOVJ EC00121
SMOVL C00122 +MOVJ EC00122
SMOVL C00123 +MOVJ EC00123
SMOVL C00124 +MOVJ EC00124
SMOVL C00125 +MOVJ EC00125
SMOVL C00126 +MOVJ EC00126
SMOVL C00127 +MOVJ EC00127
SMOVL C00128 +MOVJ EC00128
SMOVL C00129 +MOVJ EC00129
SMOVL C00130 +MOVJ EC00130
SMOVL C00131 +MOVJ EC00131
SMOVL C00132 +MOVJ EC00132
SMOVL C00133 +MOVJ EC00133
SMOVL C00134 +MOVJ EC00134
SMOVL C00135 +MOVJ EC00135
SMOVL C00136 +MOVJ EC00136
SMOVL C00137 +MOVJ EC00137
SMOVL C00138 +MOVJ EC00138
SMOVL C00139 +MOVJ EC00139
SMOVL C00140 +MOVJ EC00140
SMOVL C00141 +MOVJ EC00141
SMOVL C00142 +MOVJ EC00142
SMOVL C00143 +MOVJ EC00143
SMOVL C00144 +MOVJ EC00144
SMOVL C00145 +MOVJ EC00145
SMOVL C00146 +MOVJ EC00146
SMOVL C00147 +MOVJ EC00147
SMOVL C00148 +MOVJ EC00148
SMOVL C00149 +MOVJ EC00149
SMOVL C00150 +MOVJ EC00150
SMOVL C00151 +MOVJ EC00151
SMOVL C00152 +MOVJ EC00152
SMOVL C00153 +MOVJ EC00153
SMOVL C00154 +MOVJ EC00154
SMOVL C00155 +MOVJ EC00155
SMOVL C00156 +MOVJ EC00156
SMOVL C00157 +MOVJ EC00157
SMOVL C00158 +MOVJ EC00158
SMOVL C00159 +MOVJ EC00159
SMOVL C00160 +MOVJ EC00160
SMOVL C00161 +MOVJ EC00161
SMOVL C00162 +MOVJ EC00162
SMOVL C00163 +MOVJ EC00163
SMOVL C00164 +MOVJ EC00164
SMOVL C00165 +MOVJ EC00165
SMOVL C00166 +MOVJ EC00166
SMOVL C00167 +MOVJ EC00167
SMOVL C00168 +MOVJ EC00168
SMOVL C00169 +MOVJ EC00169
SMOVL C00170 +MOVJ EC00170
SMOVL C00171 +MOVJ EC00171
SMOVL C00172 +MOVJ EC00172
SMOVL C00173 +MOVJ EC00173
SMOVL C00174 +MOVJ EC00174
SMOVL C00175 +MOVJ EC00175
SMOVL C00176 +MOVJ EC00176
SMOVL C00177 +MOVJ EC00177
SMOVL C00178 +MOVJ EC00178
SMOVL C00179 +MOVJ EC00179
SMOVL C00180 +MOVJ EC00180
SMOVL C00181 +MOVJ EC00181
SMOVL C00182 +MOVJ EC00182
SMOVL C00183 +MOVJ EC00183
SMOVL C00184 +MOVJ EC00184
SMOVL C00185 +MOVJ EC00185
SMOVL C00186 +MOVJ EC00186
SMOVL C00187 +MOVJ EC00187
SMOVL C00188 +MOVJ EC00188
SMOVL C00189 +MOVJ EC00189
SMOVL C00190 +MOVJ EC00190
SMOVL C00191 +MOVJ EC00191
SMOVL C00192 +MOVJ EC00192
SMOVL C00193 +MOVJ EC00193
SMOVL C00194 +MOVJ EC00194
SMOVL C00195 +MOVJ EC00195
SMOVL C00196 +MOVJ EC00196
SMOVL C00197 +MOVJ EC00197
SMOVL C00198 +MOVJ EC00198
SMOVL C00199 +MOVJ EC00199
SMOVL C00200 +MOVJ EC00200
SMOVL C00201 +MOVJ EC00201
SMOVL C00202 +MOVJ EC00202
SMOVL C00203 +MOVJ EC00203
SMOVL C00204 +MOVJ EC00204
SMOVL C00205 +MOVJ EC00205
SMOVL C00206 +MOVJ EC00206
SMOVL C00207 +MOVJ EC00207
SMOVL C00208 +MOVJ EC00208
SMOVL C00209 +MOVJ EC00209
SMOVL C00210 +MOVJ EC00210
SMOVL C00211 +MOVJ EC00211
SMOVL C00212 +MOVJ EC00212
SMOVL C00213 +MOVJ EC00213
SMOVL C00214 +MOVJ EC00214
SMOVL C00215 +MOVJ EC00215
SMOVL C00216 +MOVJ EC00216
SMOVL C00217 +MOVJ EC00217
SMOVL C00218 +MOVJ EC00218
SMOVL C00219 +MOVJ EC00219
SMOVL C00220 +MOVJ EC00220
SMOVL C00221 +MOVJ EC00221
SMOVL C00222 +MOVJ EC00222
SMOVL C00223 +MOVJ EC00223
SMOVL C00224 +MOVJ EC00224
SMOVL C00225 +MOVJ EC00225
SMOVL C00226 +MOVJ EC00226
SMOVL C00227 +MOVJ EC00227
SMOVL C00228 +MOVJ EC00228
SMOVL C00229 +MOVJ EC00229
SMOVL C00230 +MOVJ EC00230
SMOVL C00231 +MOVJ EC00231
SMOVL C00232 +MOVJ EC00232
SMOVL C00233 +MOVJ EC00233
SMOVL C00234 +MOVJ EC00234
SMOVL C00235 +MOVJ EC00235
SMOVL C00236 +MOVJ EC00236
SMOVL C00237 +MOVJ EC00237
SMOVL C00238 +MOVJ EC00238
SMOVL C00239 +MOVJ EC00239
SMOVL C00240 +MOVJ EC00240
SMOVL C00241 +MOVJ EC00241
SMOVL C00242 +MOVJ EC00242
SMOVL C00243 +MOVJ EC00243
SMOVL C00244 +MOVJ EC00244
SMOVL C00245 +MOVJ EC00245
SMOVL C00246 +MOVJ EC00246
SMOVL C00247 +MOVJ EC00247
SMOVL C00248 +MOVJ EC00248
SMOVL C00249 +MOVJ EC00249
SMOVL C00250 +MOVJ EC00250
SMOVL C00251 +MOVJ EC00251
SMOVL C00252 +MOVJ EC00252
SMOVL C00253 +MOVJ EC00253
SMOVL C00254 +MOVJ EC00254
SMOVL C00255 +MOVJ EC00255
SMOVL C00256 +MOVJ EC00256
SMOVL C00257 +MOVJ EC00257
SMOVL C00258 +MOVJ EC00258
SMOVL C00259 +MOVJ EC00259
SMOVL C00260 +MOVJ EC00260
SMOVL C00261 +MOVJ EC00261
SMOVL C00262 +MOVJ EC00262
SMOVL C00263 +MOVJ EC00263
SMOVL C00264 +MOVJ EC00264
SMOVL C00265 +MOVJ EC00265
SMOVL C00266 +MOVJ EC00266
SMOVL C00267 +MOVJ EC00267
SMOVL C00268 +MOVJ EC00268
SMOVL C00269 +MOVJ EC00269
SMOVL C00270 +MOVJ EC00270
SMOVL C00271 +MOVJ EC00271
SMOVL C00272 +MOVJ EC00272
SMOVL C00273 +MOVJ EC00273
SMOVL C00274 +MOVJ EC00274
SMOVL C00275 +MOVJ EC00275
SMOVL C00276 +MOVJ EC00276
SMOVL C00277 +MOVJ EC00277
SMOVL C00278 +MOVJ EC00278
SMOVL C00279 +MOVJ EC00279
SMOVL C00280 +MOVJ EC00280
SMOVL C00281 +MOVJ EC00281
SMOVL C00282 +MOVJ EC00282
SMOVL C00283 +MOVJ EC00283
SMOVL C00284 +MOVJ EC00284
SMOVL C00285 +MOVJ EC00285
SMOVL C00286 +MOVJ EC00286
SMOVL C00287 +MOVJ EC00287
SMOVL C00288 +MOVJ EC00288
SMOVL C00289 +MOVJ EC00289
SMOVL C00290 +MOVJ EC00290
SMOVL C00291 +MOVJ EC00291
SMOVL C00292 +MOVJ EC00292
SMOVL C00293 +MOVJ EC00293
SMOVL C00294 +MOVJ EC00294
SMOVL C00295 +MOVJ EC00295
SMOVL C00296 +MOVJ EC00296
SMOVL C00297 +MOVJ EC00297
SMOVL C00298 +MOVJ EC00298
SMOVL C00299 +MOVJ EC00299
SMOVL C00300 +MOVJ EC00300
SMOVL C00301 +MOVJ EC00301
SMOVL C00302 +MOVJ EC00302
SMOVL C00303 +MOVJ EC00303
SMOVL C00304 +MOVJ EC00304
SMOVL C00305 +MOVJ EC00305
SMOVL C00306 +MOVJ EC00306
SMOVL C00307 +MOVJ EC00307
SMOVL C00308 +MOVJ EC00308
SMOVL C00309 +MOVJ EC00309
SMOVL C00310 +MOVJ EC00310
SMOVL C00311 +MOVJ EC00311
SMOVL C00312 +MOVJ EC00312
SMOVL C00313 +MOVJ EC00313
SMOVL C00314 +MOVJ EC00314
SMOVL C00315 +MOVJ EC00315
SMOVL C00316 +MOVJ EC00316
SMOVL C00317 +MOVJ EC00317
SMOVL C00318 +MOVJ EC00318
SMOVL C00319 +MOVJ EC00319
SMOVL C00320 +MOVJ EC00320
SMOVL C00321 +MOVJ EC00321
SMOVL C00322 +MOVJ EC00322
SMOVL C00323 +MOVJ EC00323
SMOVL C00324 +MOVJ EC00324
SMOVL C00325 +MOVJ EC00325
SMOVL C00326 +MOVJ EC00326
SMOVL C00327 +MOVJ EC00327
SMOVL C00328 +MOVJ EC00328
SMOVL C00329 +MOVJ EC00329
SMOVL C00330 +MOVJ EC00330
SMOVL C00331 +MOVJ EC00331
SMOVL C00332 +MOVJ EC00332
SMOVL C00333 +MOVJ EC00333
SMOVL C00334 +MOVJ EC00334
SMOVL C00335 +MOVJ EC00335
SMOVL C00336 +MOVJ EC00336
SMOVL C00337 +MOVJ EC00337
SMOVL C00338 +MOVJ EC00338
SMOVL C00339 +MOVJ EC00339
SMOVL C00340 +MOVJ EC00340
SMOVL C00341 +MOVJ EC00341
SMOVL C00342 +MOVJ EC00342
SMOVL C00343 +MOVJ EC00343
SMOVL C00344 +MOVJ EC00344
SMOVL C00345 +MOVJ EC00345
SMOVL C00346 +MOVJ EC00346
SMOVL C00347 +MOVJ EC00347
SMOVL C00348 +MOVJ EC00348
SMOVL C00349 +MOVJ EC00349
SMOVL C00350 +MOVJ EC00350
SMOVL C00351 +MOVJ EC00351
SMOVL C00352 +MOVJ EC00352
SMOVL C00353 +MOVJ EC00353
SMOVL C00354 +MOVJ EC00354
SMOVL C00355 +MOVJ EC00355
SMOVL C00356 +MOVJ EC00356
SMOVL C00357 +MOVJ EC00357
SMOVL C00358 +MOVJ EC00358
SMOVL C00359 +MOVJ EC00359
SMOVL C00360 +MOVJ EC00360
SMOVL C00361 +MOVJ EC00361
SMOVL C00362 +MOVJ EC00362
SMOVL C00363 +MOVJ EC00363
SMOVL C00364 +MOVJ EC00364
SMOVL C00365 +MOVJ EC00365
SMOVL C00366 +MOVJ EC00366
SMOVL C00367 +MOVJ EC00367
SMOVL C00368 +MOVJ EC00368
SMOVL C00369 +MOVJ EC00369
SMOVL C00370 +MOVJ EC00370
SMOVL C00371 +MOVJ EC00371
SMOVL C00372 +MOVJ EC00372
SMOVL C00373 +MOVJ EC00373
SMOVL C00374 +MOVJ EC00374
SMOVL C00375 +MOVJ EC00375
SMOVL C00376 +MOVJ EC00376
SMOVL C00377 +MOVJ EC00377
SMOVL C00378 +MOVJ EC00378
SMOVL C00379 +MOVJ EC00379
SMOVL C00380 +MOVJ EC00380
SMOVL C00381 +MOVJ EC00381
SMOVL C00382 +MOVJ EC00382
SMOVL C00383 +MOVJ EC00383
SMOVL C00384 +MOVJ EC00384
SMOVL C00385 +MOVJ EC00385
SMOVL C00386 +MOVJ EC00386
SMOVL C00387 +MOVJ EC00387
SMOVL C00388 +MOVJ EC00388
SMOVL C00389 +MOVJ EC00389
SMOVL C00390 +MOVJ EC00390
SMOVL C00391 +MOVJ EC00391
SMOVL C00392 +MOVJ EC00392
SMOVL C00393 +MOVJ EC00393
SMOVL C00394 +MOVJ EC00394
SMOVL C00395 +MOVJ EC00395
SMOVL C00396 +MOVJ EC00396
SMOVL C00397 +MOVJ EC00397
SMOVL C00398 +MOVJ EC00398
SMOVL C00399 +MOVJ EC00399
SMOVL C00400 +MOVJ EC00400
SMOVL C00401 +MOVJ EC00401
SMOVL C00402 +MOVJ EC00402
SMOVL C00403 +MOVJ EC00403
SMOVL C00404 +MOVJ EC00404
SMOVL C00405 +MOVJ EC00405
SMOVL C00406 +MOVJ EC00406
SMOVL C00407 +MOVJ EC00407
SMOVL C00408 +MOVJ EC00408
SMOVL C00409 +MOVJ EC00409
SMOVL C00410 +MOVJ EC00410
SMOVL C00411 +MOVJ EC00411
SMOVL C00412 +MOVJ EC00412
SMOVL C00413 +MOVJ EC00413
SMOVL C00414 +MOVJ EC00414
SMOVL C00415 +MOVJ EC00415
SMOVL C00416 +MOVJ EC00416
SMOVL C00417 +MOVJ EC00417
SMOVL C00418 +MOVJ EC00418
SMOVL C00419 +MOVJ EC00419
SMOVL C00420 +MOVJ EC00420
SMOVL C00421 +MOVJ EC00421
SMOVL C00422 +MOVJ EC00422
SMOVL C00423 +MOVJ EC00423
SMOVL C00424 +MOVJ EC00424
SMOVL C00425 +MOVJ EC00425
SMOVL C00426 +MOVJ EC00426
SMOVL C00427 +MOVJ EC00427
SMOVL C00428 +MOVJ EC00428
SMOVL C00429 +MOVJ EC00429
SMOVL C00430 +MOVJ EC00430
SMOVL C00431 +MOVJ EC00431
SMOVL C00432 +MOVJ EC00432
SMOVL C00433 +MOVJ EC00433
SMOVL C00434 +MOVJ EC00434
SMOVL C00435 +MOVJ EC00435
SMOVL C00436 +MOVJ EC00436
SMOVL C00437 +MOVJ EC00437
SMOVL C00438 +MOVJ EC00438
SMOVL C00439 +MOVJ EC00439
SMOVL C00440 +MOVJ EC00440
SMOVL C00441 +MOVJ EC00441
SMOVL C00442 +MOVJ EC00442
SMOVL C00443 +MOVJ EC00443
SMOVL C00444 +MOVJ EC00444
SMOVL C00445 +MOVJ EC00445
SMOVL C00446 +MOVJ EC00446
SMOVL C00447 +MOVJ EC00447
SMOVL C00448 +MOVJ EC00448
SMOVL C00449 +MOVJ EC00449
SMOVL C00450 +MOVJ EC00450
SMOVL C00451 +MOVJ EC00451
SMOVL C00452 +MOVJ EC00452
SMOVL C00453 +MOVJ EC00453
SMOVL C00454 +MOVJ EC00454
SMOVL C00455 +MOVJ EC00455
SMOVL C00456 +MOVJ EC00456
SMOVL C00457 +MOVJ EC00457
SMOVL C00458 +MOVJ EC00458
SMOVL C00459 +MOVJ EC00459
SMOVL C00460 +MOVJ EC00460
SMOVL C00461 +MOVJ EC00461
SMOVL C00462 +MOVJ EC00462
SMOVL C00463 +MOVJ EC00463
SMOVL C00464 +MOVJ EC00464
SMOVL C00465 +MOVJ EC00465
SMOVL C00466 +MOVJ EC00466
SMOVL C00467 +MOVJ EC00467
SMOVL C00468 +MOVJ EC00468
SMOVL C00469 +MOVJ EC00469
SMOVL C00470 +MOVJ EC00470
SMOVL C00471 +MOVJ EC00471
SMOVL C00472 +MOVJ EC00472
SMOVL C00473 +MOVJ EC00473
SMOVL C00474 +MOVJ EC00474
SMOVL C00475 +MOVJ EC00475
SMOVL C00476 +MOVJ EC00476
SMOVL C00477 +MOVJ EC00477
SMOVL C00478 +MOVJ EC00478
SMOVL C00479 +MOVJ EC00479
SMOVL C00480 +MOVJ EC00480
SMOVL C00481 +MOVJ EC00481
SMOVL C00482 +MOVJ EC00482
SMOVL C00483 +MOVJ EC00483
SMOVL C00484 +MOVJ EC00484
SMOVL C00485 +MOVJ EC00485
SMOVL C00486 +MOVJ EC00486
SMOVL C00487 +MOVJ EC00487
SMOVL C00488 +MOVJ EC00488
SMOVL C00489 +MOVJ EC00489
SMOVL C00490 +MOVJ EC00490
SMOVL C00491 +MOVJ EC00491
SMOVL C00492 +MOVJ EC00492
SMOVL C00493 +MOVJ EC00493
SMOVL C00494 +MOVJ EC00494
SMOVL C00495 +MOVJ EC00495
SMOVL C00496 +MOVJ EC00496
SMOVL C00497 +MOVJ EC00497
SMOVL C00498 +MOVJ EC00498
SMOVL C00499 +MOVJ EC00499
SMOVL C00500 +MOVJ EC00500
SMOVL C00501 +MOVJ EC00501
SMOVL C00502 +MOVJ EC00502
SMOVL C00503 +MOVJ EC00503
SMOVL C00504 +MOVJ EC00504
SMOVL C00505 +MOVJ EC00505
SMOVL C00506 +MOVJ EC00506
SMOVL C00507 +MOVJ EC00507
SMOVL C00508 +MOVJ EC00508
SMOVL C00509 +MOVJ EC00509
SMOVL C00510 +MOVJ EC00510
SMOVL C00511 +MOVJ EC00511
SMOVL C00512 +MOVJ EC00512
SMOVL C00513 +MOVJ EC00513
SMOVL C00514 +MOVJ EC00514
SMOVL C00515 +MOVJ EC00515
SMOVL C00516 +MOVJ EC00516
SMOVL C00517 +MOVJ EC00517
SMOVL C00518 +MOVJ EC00518
SMOVL C00519 +MOVJ EC00519
SMOVL C00520 +MOVJ EC00520
SMOVL C00521 +MOVJ EC00521
SMOVL C00522 +MOVJ EC00522
SMOVL C00523 +MOVJ EC00523
SMOVL C00524 +MOVJ EC00524
SMOVL C00525 +MOVJ EC00525
SMOVL C00526 +MOVJ EC00526
SMOVL C00527 +MOVJ EC00527
SMOVL C00528 +MOVJ EC00528
SMOVL C00529 +MOVJ EC00529
SMOVL C00530 +MOVJ EC00530
SMOVL C00531 +MOVJ EC00531
SMOVL C00532 +MOVJ EC00532
SMOVL C00533 +MOVJ EC00533
SMOVL C00534 +MOVJ EC00534
SMOVL C00535 +MOVJ EC00535
SMOVL C00536 +MOVJ EC00536
SMOVL C00537 +MOVJ EC00537
SMOVL C00538 +MOVJ EC00538
SMOVL C00539 +MOVJ EC00539
SMOVL C00540 +MOVJ EC00540
SMOVL C00541 +MOVJ EC00541
SMOVL C00542 +MOVJ EC00542
SMOVL C00543 +MOVJ EC00543
SMOVL C00544 +MOVJ EC00544
SMOVL C00545 +MOVJ EC00545
SMOVL C00546 +MOVJ EC00546
SMOVL C00547 +MOVJ EC00547
SMOVL C00548 +MOVJ EC00548
SMOVL C00549 +MOVJ EC00549
SMOVL C00550 +MOVJ EC00550
SMOVL C00551 +MOVJ EC00551
SMOVL C00552 +MOVJ EC00552
SMOVL C00553 +MOVJ EC00553
SMOVL C00554 +MOVJ EC00554
SMOVL C00555 +MOVJ EC00555
SMOVL C00556 +MOVJ EC00556
SMOVL C00557 +MOVJ EC00557
SMOVL C00558 +MOVJ EC00558
SMOVL C00559 +MOVJ EC00559
SMOVL C00560 +MOVJ EC00560
SMOVL C00561 +MOVJ EC00561
SMOVL C00562 +MOVJ EC00562
SMOVL C00563 +MOVJ EC00563
SMOVL C00564 +MOVJ EC00564
SMOVL C00565 +MOVJ EC00565
SMOVL C00566 +MOVJ EC00566
SMOVL C00567 +MOVJ EC00567
SMOVL C00568 +MOVJ EC00568
SMOVL C00569 +MOVJ EC00569
SMOVL C00570 +MOVJ EC00570
SMOVL C00571 +MOVJ EC00571
SMOVL C00572 +MOVJ EC00572
SMOVL C00573 +MOVJ EC00573
SMOVL C00574 +MOVJ EC00574
SMOVL C00575 +MOVJ EC00575
SMOVL C00576 +MOVJ EC00576
SMOVL C00577 +MOVJ EC00577
SMOVL C00578 +MOVJ EC00578
SMOVL C00579 +MOVJ EC00579
SMOVL C00580 +MOVJ EC00580
SMOVL C00581 +MOVJ EC00581
SMOVL C00582 +MOVJ EC00582
SMOVL C00583 +MOVJ EC00583
SMOVL C00584 +MOVJ EC00584
SMOVL C00585 +MOVJ EC00585
SMOVL C00586 +MOVJ EC00586
SMOVL C00587 +MOVJ EC00587
SMOVL C00588 +MOVJ EC00588
SMOVL C00589 +MOVJ EC00589
SMOVL C00590 +MOVJ EC00590
SMOVL C00591 +MOVJ EC00591
SMOVL C00592 +MOVJ EC00592
SMOVL C00593 +MOVJ EC00593
SMOVL C00594 +MOVJ EC00594
SMOVL C00595 +MOVJ EC00595
SMOVL C00596 +MOVJ EC00596
SMOVL C00597 +MOVJ EC00597
SMOVL C00598 +MOVJ EC00598
SMOVL C00599 +MOVJ EC00599
SMOVL C00600 +MOVJ EC00600
SMOVL C00601 +MOVJ EC00601
SMOVL C00602 +MOVJ EC00602
SMOVL C00603 +MOVJ EC00603
SMOVL C00604 +MOVJ EC00604
SMOVL C00605 +MOVJ EC00605
SMOVL C00606 +MOVJ EC00606
SMOVL C00607 +MOVJ EC00607
SMOVL C00608 +MOVJ EC00608
SMOVL C00609 +MOVJ EC00609
SMOVL C00610 +MOVJ EC00610
SMOVL C00611 +MOVJ EC00611
SMOVL C00612 +MOVJ EC00612
SMOVL C00613 +MOVJ EC00613
SMOVL C00614 +MOVJ EC00614
SMOVL C00615 +MOVJ EC00615
SMOVL C00616 +MOVJ EC00616
SMOVL C00617 +MOVJ EC00617
SMOVL C00618 +MOVJ EC00618
SMOVL C00619 +MOVJ EC00619
SMOVL C00620 +MOVJ EC00620
SMOVL C00621 +MOVJ EC00621
SMOVL C00622 +MOVJ EC00622
SMOVL C00623 +MOVJ EC00623
SMOVL C00624 +MOVJ EC00624
SMOVL C00625 +MOVJ EC00625
SMOVL C00626 +MOVJ EC00626
SMOVL C00627 +MOVJ EC00627
SMOVL C00628 +MOVJ EC00628
SMOVL C00629 +MOVJ EC00629
SMOVL C00630 +MOVJ EC00630
SMOVL C00631 +MOVJ EC00631
SMOVL C00632 +MOVJ EC00632
SMOVL C00633 +MOVJ EC00633
SMOVL C00634 +MOVJ EC00634
SMOVL C00635 +MOVJ EC00635
SMOVL C00636 +MOVJ EC00636
SMOVL C00637 +MOVJ EC00637
SMOVL C00638 +MOVJ EC00638
SMOVL C00639 +MOVJ EC00639
SMOVL C00640 +MOVJ EC00640
SMOVL C00641 +MOVJ EC00641
SMOVL C00642 +MOVJ EC00642
SMOVL C00643 +MOVJ EC00643
SMOVL C00644 +MOVJ EC00644
SMOVL C00645 +MOVJ EC00645
SMOVL C00646 +MOVJ EC00646
SMOVL C00647 +MOVJ EC00647
SMOVL C00648 +MOVJ EC00648
SMOVL C00649 +MOVJ EC00649
SMOVL C00650 +MOVJ EC00650
SMOVL C00651 +MOVJ EC00651
SMOVL C00652 +MOVJ EC00652
SMOVL C00653 +MOVJ EC00653
SMOVL C00654 +MOVJ EC00654
SMOVL C00655 +MOVJ EC00655
SMOVL C00656 +MOVJ EC00656
SMOVL C00657 +MOVJ EC00657
SMOVL C00658 +MOVJ EC00658
SMOVL C00659 +MOVJ EC00659
SMOVL C00660 +MOVJ EC00660
SMOVL C00661 +MOVJ EC00661
SMOVL C00662 +MOVJ EC00662
SMOVL C00663 +MOVJ EC00663
SMOVL C00664 +MOVJ EC00664
SMOVL C00665 +MOVJ EC00665
SMOVL C00666 +MOVJ EC00666
SMOVL C00667 +MOVJ EC00667
SMOVL C00668 +MOVJ EC00668
SMOVL C00669 +MOVJ EC00669
SMOVL C00670 +MOVJ EC00670
SMOVL C00671 +MOVJ EC00671
SMOVL C00672 +MOVJ EC00672
SMOVL C00673 +MOVJ EC00673
SMOVL C00674 +MOVJ EC00674
SMOVL C00675 +MOVJ EC00675
SMOVL C00676 +MOVJ EC00676
SMOVL C00677 +MOVJ EC00677
SMOVL C00678 +MOVJ EC00678
SMOVL C00679 +MOVJ EC00679
SMOVL C00680 +MOVJ EC00680
SMOVL C00681 +MOVJ EC00681
SMOVL C00682 +MOVJ EC00682
SMOVL C00683 +MOVJ EC00683
SMOVL C00684 +MOVJ EC00684
SMOVL C00685 +MOVJ EC00685
SMOVL C00686 +MOVJ EC00686
SMOVL C00687 +MOVJ EC00687
SMOVL C00688 +MOVJ EC00688
SMOVL C00689 +MOVJ EC00689
SMOVL C00690 +MOVJ EC00690
SMOVL C00691 +MOVJ EC00691
SMOVL C00692 +MOVJ EC00692
SMOVL C00693 +MOVJ EC00693
SMOVL C00694 +MOVJ EC00694
SMOVL C00695 +MOVJ EC00695
SMOVL C00696 +MOVJ EC00696
SMOVL C00697 +MOVJ EC00697
SMOVL C00698 +MOVJ EC00698
SMOVL C00699 +MOVJ EC00699
SMOVL C00700 +MOVJ EC00700
SMOVL C00701 +MOVJ EC00701
SMOVL C00702 +MOVJ EC00702
SMOVL C00703 +MOVJ EC00703
SMOVL C00704 +MOVJ EC00704
SMOVL C00705 +MOVJ EC00705
SMOVL C00706 +MOVJ EC00706
SMOVL C00707 +MOVJ EC00707
SMOVL C00708 +MOVJ EC00708
SMOVL C00709 +MOVJ EC00709
SMOVL C00710 +MOVJ EC00710
SMOVL C00711 +MOVJ EC00711
SMOVL C00712 +MOVJ EC00712
SMOVL C00713 +MOVJ EC00713
SMOVL C00714 +MOVJ EC00714
SMOVL C00715 +MOVJ EC00715
SMOVL C00716 +MOVJ EC00716
SMOVL C00717 +MOVJ EC00717
SMOVL C00718 +MOVJ EC00718
SMOVL C00719 +MOVJ EC00719
SMOVL C00720 +MOVJ EC00720
SMOVL C00721 +MOVJ EC00721
SMOVL C00722 +MOVJ EC00722
SMOVL C00723 +MOVJ EC00723
SMOVL C00724 +MOVJ EC00724
SMOVL C00725 +MOVJ EC00725
SMOVL C00726 +MOVJ EC00726
SMOVL C00727 +MOVJ EC00727
SMOVL C00728 +MOVJ EC00728
SMOVL C00729 +MOVJ EC00729
SMOVL C00730 +MOVJ EC00730
SMOVL C00731 +MOVJ EC00731
SMOVL C00732 +MOVJ EC00732
SMOVL C00733 +MOVJ EC00733
SMOVL C00734 +MOVJ EC00734
SMOVL C00735 +MOVJ EC00735
SMOVL C00736 +MOVJ EC00736
SMOVL C00737 +MOVJ EC00737
SMOVL C00738 +MOVJ EC00738
SMOVL C00739 +MOVJ EC00739
SMOVL C00740 +MOVJ EC00740
SMOVL C00741 +MOVJ EC00741
SMOVL C00742 +MOVJ EC00742
SMOVL C00743 +MOVJ EC00743
SMOVL C00744 +MOVJ EC00744
SMOVL C00745 +MOVJ EC00745
SMOVL C00746 +MOVJ EC00746
SMOVL C00747 +MOVJ EC00747
SMOVL C00748 +MOVJ EC00748
SMOVL C00749 +MOVJ EC00749
SMOVL C00750 +MOVJ EC00750
SMOVL C00751 +MOVJ EC00751
SMOVL C00752 +MOVJ EC00752
SMOVL C00753 +MOVJ EC00753
SMOVL C00754 +MOVJ EC00754
SMOVL C00755 +MOVJ EC00755
SMOVL C00756 +MOVJ EC00756
SMOVL C00757 +MOVJ EC00757
SMOVL C00758 +MOVJ EC00758
SMOVL C00759 +MOVJ EC00759
SMOVL C00760 +MOVJ EC00760
SMOVL C00761 +MOVJ EC00761
SMOVL C00762 +MOVJ EC00762
SMOVL C00763 +MOVJ EC00763
SMOVL C00764 +MOVJ EC00764
SMOVL C00765 +MOVJ EC00765
SMOVL C00766 +MOVJ EC00766
SMOVL C00767 +MOVJ EC00767
SMOVL C00768 +MOVJ EC00768
SMOVL C00769 +MOVJ EC00769
SMOVL C00770 +MOVJ EC00770
SMOVL C00771 +MOVJ EC00771
SMOVL C00772 +MOVJ EC00772
SMOVL C00773 +MOVJ EC00773
SMOVL C00774 +MOVJ EC00774
SMOVL C00775 +MOVJ EC00775
SMOVL C00776 +MOVJ EC00776
SMOVL C00777 +MOVJ EC00777
SMOVL C00778 +MOVJ EC00778
SMOVL C00779 +MOVJ EC00779
SMOVL C00780 +MOVJ EC00780
SMOVL C00781 +MOVJ EC00781
SMOVL C00782 +MOVJ EC00782
SMOVL C00783 +MOVJ EC00783
SMOVL C00784 +MOVJ EC00784
SMOVL C00785 +MOVJ EC00785
SMOVL C00786 +MOVJ EC00786
SMOVL C00787 +MOVJ EC00787
SMOVL C00788 +MOVJ EC00788
SMOVL C00789 +MOVJ EC00789
SMOVL C00790 +MOVJ EC00790
SMOVL C00791 +MOVJ EC00791
SMOVL C00792 +MOVJ EC00792
SMOVL C00793 +MOVJ EC00793
SMOVL C00794 +MOVJ EC00794
SMOVL C00795 +MOVJ EC00795
SMOVL C00796 +MOVJ EC00796
SMOVL C00797 +MOVJ EC00797
SMOVL C00798 +MOVJ EC00798
SMOVL C00799 +MOVJ EC00799
SMOVL C00800 +MOVJ EC00800
SMOVL C00801 +MOVJ EC00801
SMOVL C00802 +MOVJ EC00802
SMOVL C00803 +MOVJ EC00803
SMOVL C00804 +MOVJ EC00804
SMOVL C00805 +MOVJ EC00805
SMOVL C00806 +MOVJ EC00806
SMOVL C00807 +MOVJ EC00807
SMOVL C00808 +MOVJ EC00808
SMOVL C00809 +MOVJ EC00809
SMOVL C00810 +MOVJ EC00810
SMOVL C00811 +MOVJ EC00811
SMOVL C00812 +MOVJ EC00812
SMOVL C00813 +MOVJ EC00813
SMOVL C00814 +MOVJ EC00814
SMOVL C00815 +MOVJ EC00815
SMOVL C00816 +MOVJ EC00816
SMOVL C00817 +MOVJ EC00817
SMOVL C00818 +MOVJ EC00818
SMOVL C00819 +MOVJ EC00819
SMOVL C00820 +MOVJ EC00820
SMOVL C00821 +MOVJ EC00821
SMOVL C00822 +MOVJ EC00822
SMOVL C00823 +MOVJ EC00823
SMOVL C00824 +MOVJ EC00824
SMOVL C00825 +MOVJ EC00825
SMOVL C00826 +MOVJ EC00826
SMOVL C00827 +MOVJ EC00827
SMOVL C00828 +MOVJ EC00828
SMOVL C00829 +MOVJ EC00829
SMOVL C00830 +MOVJ EC00830
SMOVL C00831 +MOVJ EC00831
SMOVL C00832 +MOVJ EC00832
SMOVL C00833 +MOVJ EC00833
SMOVL C00834 +MOVJ EC00834
SMOVL C00835 +MOVJ EC00835
SMOVL C00836 +MOVJ EC00836
SMOVL C00837 +MOVJ EC00837
SMOVL C00838 +MOVJ EC00838
SMOVL C00839 +MOVJ EC00839
SMOVL C00840 +MOVJ EC00840
SMOVL C00841 +MOVJ EC00841
SMOVL C00842 +MOVJ EC00842
SMOVL C00843 +MOVJ EC00843
SMOVL C00844 +MOVJ EC00844
SMOVL C00845 +MOVJ EC00845
SMOVL C00846 +MOVJ EC00846
SMOVL C00847 +MOVJ EC00847
SMOVL C00848 +MOVJ EC00848
SMOVL C00849 +MOVJ EC00849
SMOVL C00850 +MOVJ EC00850
SMOVL C00851 +MOVJ EC00851
SMOVL C00852 +MOVJ EC00852
SMOVL C00853 +MOVJ EC00853
SMOVL C00854 +MOVJ EC00854
SMOVL C00855 +MOVJ EC00855
SMOVL C00856 +MOVJ EC00856
SMOVL C00857 +MOVJ EC00857
SMOVL C00858 +MOVJ EC00858
SMOVL C00859 +MOVJ EC00859
SMOVL C00860 +MOVJ EC00860
SMOVL C00861 +MOVJ EC00861
SMOVL C00862 +MOVJ EC00862
SMOVL C00863 +MOVJ EC00863
SMOVL C00864 +MOVJ EC00864
SMOVL C00865 +MOVJ EC00865
SMOVL C00866 +MOVJ EC00866
SMOVL C00867 +MOVJ EC00867
SMOVL C00868 +MOVJ EC00868
SMOVL C00869 +MOVJ EC00869
SMOVL C00870 +MOVJ EC00870
SMOVL C00871 +MOVJ EC00871
SMOVL C00872 +MOVJ EC00872
SMOVL C00873 +MOVJ EC00873
SMOVL C00874 +MOVJ EC00874
SMOVL C00875 +MOVJ EC00875
SMOVL C00876 +MOVJ EC00876
SMOVL C00877 +MOVJ EC00877
SMOVL C00878 +MOVJ EC00878
SMOVL C00879 +MOVJ EC00879
SMOVL C00880 +MOVJ EC00880
SMOVL C00881 +MOVJ EC00881
SMOVL C00882 +MOVJ EC00882
SMOVL C00883 +MOVJ EC00883
SMOVL C00884 +MOVJ EC00884
SMOVL C00885 +MOVJ EC00885
SMOVL C00886 +MOVJ EC00886
SMOVL C00887 +MOVJ EC00887
SMOVL C00888 +MOVJ EC00888
SMOVL C00889 +MOVJ EC00889
SMOVL C00890 +MOVJ EC00890
SMOVL C00891 +MOVJ EC00891
SMOVL C00892 +MOVJ EC00892
SMOVL C00893 +MOVJ EC00893
SMOVL C00894 +MOVJ EC00894
SMOVL C00895 +MOVJ EC00895
SMOVL C00896 +MOVJ EC00896
SMOVL C00897 +MOVJ EC00897
SMOVL C00898 +MOVJ EC00898
SMOVL C00899 +MOVJ EC00899
SMOVL C00900 +MOVJ EC00900
SMOVL C00901 +MOVJ EC00901
SMOVL C00902 +MOVJ EC00902
SMOVL C00903 +MOVJ EC00903
SMOVL C00904 +MOVJ EC00904
SMOVL C00905 +MOVJ EC00905
SMOVL C00906 +MOVJ EC00906
SMOVL C00907 +MOVJ EC00907
SMOVL C00908 +MOVJ EC00908
SMOVL C00909 +MOVJ EC00909
SMOVL C00910 +MOVJ EC00910
SMOVL C00911 +MOVJ EC00911
SMOVL C00912 +MOVJ EC00912
SMOVL C00913 +MOVJ EC00913
SMOVL C00914 +MOVJ EC00914
SMOVL C00915 +MOVJ EC00915
SMOVL C00916 +MOVJ EC00916
SMOVL C00917 +MOVJ EC00917
SMOVL C00918 +MOVJ EC00918
SMOVL C00919 +MOVJ EC00919
SMOVL C00920 +MOVJ EC00920
SMOVL C00921 +MOVJ EC00921
SMOVL C00922 +MOVJ EC00922
SMOVL C00923 +MOVJ EC00923
SMOVL C00924 +MOVJ EC00924
SMOVL C00925 +MOVJ EC00925
SMOVL C00926 +MOVJ EC00926
SMOVL C00927 +MOVJ EC00927
SMOVL C00928 +MOVJ EC00928
SMOVL C00929 +MOVJ EC00929
SMOVL C00930 +MOVJ EC00930
SMOVL C00931 +MOVJ EC00931
SMOVL C00932 +MOVJ EC00932
SMOVL C00933 +MOVJ EC00933
SMOVL C00934 +MOVJ EC00934
SMOVL C00935 +MOVJ EC00935
SMOVL C00936 +MOVJ EC00936
SMOVL C00937 +MOVJ EC00937
SMOVL C00938 +MOVJ EC00938
SMOVL C00939 +MOVJ EC00939
SMOVL C00940 +MOVJ EC00940
SMOVL C00941 +MOVJ EC00941
SMOVL C00942 +MOVJ EC00942
SMOVL C00943 +MOVJ EC00943
SMOVL C00944 +MOVJ EC00944
SMOVL C00945 +MOVJ EC00945
SMOVL C00946 +MOVJ EC00946
SMOVL C00947 +MOVJ EC00947
SMOVL C00948 +MOVJ EC00948
SMOVL C00949 +MOVJ EC00949
SMOVL C00950 +MOVJ EC00950
SMOVL C00951 +MOVJ EC00951
SMOVL C00952 +MOVJ EC00952
SMOVL C00953 +MOVJ EC00953
SMOVL C00954 +MOVJ EC00954
SMOVL C00955 +MOVJ EC00955
SMOVL C00956 +MOVJ EC00956
SMOVL C00957 +MOVJ EC00957
SMOVL C00958 +MOVJ EC00958
SMOVL C00959 +MOVJ EC00959
SMOVL C00960 +MOVJ EC00960
SMOVL C00961 +MOVJ EC00961
SMOVL C00962 +MOVJ EC00962
SMOVL C00963 +MOVJ EC00963
SMOVL C00964 +MOVJ EC00964
SMOVL C00965 +MOVJ EC00965
SMOVL C00966 +MOVJ EC00966
SMOVL C00967 +MOVJ EC00967
SMOVL C00968 +MOVJ EC00968
SMOVL C00969 +MOVJ EC00969
SMOVL C00970 +MOVJ EC00970
SMOVL C00971 +MOVJ EC00971
SMOVL C00972 +MOVJ EC00972
SMOVL C00973 +MOVJ EC00973
SMOVL C00974 +MOVJ EC00974
SMOVL C00975 +MOVJ EC00975
SMOVL C00976 +MOVJ EC00976
SMOVL C00977 +MOVJ EC00977
SMOVL C00978 +MOVJ EC00978
SMOVL C00979 +MOVJ EC00979
SMOVL C00980 +MOVJ EC00980
SMOVL C00981 +MOVJ EC00981
SMOVL C00982 +MOVJ EC00982
SMOVL C00983 +MOVJ EC00983
SMOVL C00984 +MOVJ EC00984
SMOVL C00985 +MOVJ EC00985
SMOVL C00986 +MOVJ EC00986
SMOVL C00987 +MOVJ EC00987
SMOVL C00988 +MOVJ EC00988
SMOVL C00989 +MOVJ EC00989
SMOVL C00990 +MOVJ EC00990
SMOVL C00991 +MOVJ EC00991
SMOVL C00992 +MOVJ EC00992
SMOVL C00993 +MOVJ EC00993
SMOVL C00994 +MOVJ EC00994
SMOVL C00995 +MOVJ EC00995
SMOVL C00996 +MOVJ EC00996
SMOVL C00997 +MOVJ EC00997
SMOVL C00998 +MOVJ EC00998
SMOVL C00999 +MOVJ EC00999
SMOVL C01000 +MOVJ EC01000
SMOVL C01001 +MOVJ EC01001
SMOVL C01002 +MOVJ EC01002
SMOVL C01003 +MOVJ EC01003
SMOVL C01004 +MOVJ EC01004
SMOVL C01005 +MOVJ EC01005
SMOVL C01006 +MOVJ EC01006
SMOVL C01007 +MOVJ EC01007
SMOVL C01008 +MOVJ EC01008
SMOVL C01009 +MOVJ EC01009
SMOVL C01010 +MOVJ EC01010
SMOVL C01011 +MOVJ EC01011
SMOVL C01012 +MOVJ EC01012
SMOVL C01013 +MOVJ EC01013
SMOVL C01014 +MOVJ EC01014
SMOVL C01015 +MOVJ EC01015
SMOVL C01016 +MOVJ EC01016
SMOVL C01017 +MOVJ EC01017
SMOVL C01018 +MOVJ EC01018
SMOVL C01019 +MOVJ EC01019
SMOVL C01020 +MOVJ EC01020
SMOVL C01021 +MOVJ EC01021
SMOVL C01022 +MOVJ EC01022
SMOVL C01023 +MOVJ EC01023
SMOVL C01024 +MOVJ EC01024
SMOVL C01025 +MOVJ EC01025
SMOVL C01026 +MOVJ EC01026
SMOVL C01027 +MOVJ EC01027
SMOVL C01028 +MOVJ EC01028
SMOVL C01029 +MOVJ EC01029
SMOVL C01030 +MOVJ EC01030
SMOVL C01031 +MOVJ EC01031
SMOVL C01032 +MOVJ EC01032
SMOVL C01033 +MOVJ EC01033
SMOVL C01034 +MOVJ EC01034
SMOVL C01035 +MOVJ EC01035
SMOVL C01036 +MOVJ EC01036
SMOVL C01037 +MOVJ EC01037
SMOVL C01038 +MOVJ EC01038
SMOVL C01039 +MOVJ EC01039
SMOVL C01040 +MOVJ EC01040
SMOVL C01041 +MOVJ EC01041
SMOVL C01042 +MOVJ EC01042
SMOVL C01043 +MOVJ EC01043
SMOVL C01044 +MOVJ EC01044
SMOVL C01045 +MOVJ EC01045
SMOVL C01046 +MOVJ EC01046
SMOVL C01047 +MOVJ EC01047
SMOVL C01048 +MOVJ EC01048
SMOVL C01049 +MOVJ EC01049
SMOVL C01050 +MOVJ EC01050
SMOVL C01051 +MOVJ EC01051
SMOVL C01052 +MOVJ EC01052
SMOVL C01053 +MOVJ EC01053
SMOVL C01054 +MOVJ EC01054
SMOVL C01055 +MOVJ EC01055
SMOVL C01056 +MOVJ EC01056
SMOVL C01057 +MOVJ EC01057
SMOVL C01058 +MOVJ EC01058
SMOVL C01059 +MOVJ EC01059
SMOVL C01060 +MOVJ EC01060
SMOVL C01061 +MOVJ EC01061
SMOVL C01062 +MOVJ EC01062
SMOVL C01063 +MOVJ EC01063
SMOVL C01064 +MOVJ EC01064
SMOVL C01065 +MOVJ EC01065
SMOVL C01066 +MOVJ EC01066
SMOVL C01067 +MOVJ EC01067
SMOVL C01068 +MOVJ EC01068
SMOVL C01069 +MOVJ EC01069
SMOVL C01070 +MOVJ EC01070
SMOVL C01071 +MOVJ EC01071
SMOVL C01072 +MOVJ EC01072
SMOVL C01073 +MOVJ EC01073
SMOVL C01074 +MOVJ EC01074
SMOVL C01075 +MOVJ EC01075
SMOVL C01076 +MOVJ EC01076
SMOVL C01077 +MOVJ EC01077
SMOVL C01078 +MOVJ EC01078
SMOVL C01079 +MOVJ EC01079
SMOVL C01080 +MOVJ EC01080
SMOVL C01081 +MOVJ EC01081
SMOVL C01082 +MOVJ EC01082
SMOVL C01083 +MOVJ EC01083
SMOVL C01084 +MOVJ EC01084
SMOVL C01085 +MOVJ EC01085
SMOVL C01086 +MOVJ EC01086
SMOVL C01087 +MOVJ EC01087
SMOVL C01088 +MOVJ EC01088
SMOVL C01089 +MOVJ EC01089
SMOVL C01090 +MOVJ EC01090
SMOVL C01091 +MOVJ EC01091
SMOVL C01092 +MOVJ EC01092
SMOVL C01093 +MOVJ EC01093
SMOVL C01094 +MOVJ EC01094
SMOVL C01095 +MOVJ EC01095
SMOVL C01096 +MOVJ EC01096
SMOVL C01097 +MOVJ EC01097
SMOVL C01098 +MOVJ EC01098
SMOVL C01099 +MOVJ EC01099
SMOVL C01100 +MOVJ EC01100
SMOVL C01101 +MOVJ EC01101
SMOVL C01102 +MOVJ EC01102
SMOVL C01103 +MOVJ EC01103
SMOVL C01104 +MOVJ EC01104
SMOVL C01105 +MOVJ EC01105
SMOVL C01106 +MOVJ EC01106
SMOVL C01107 +MOVJ EC01107
SMOVL C01108 +MOVJ EC01108
SMOVL C01109 +MOVJ EC01109
SMOVL C01110 +MOVJ EC01110
SMOVL C01111 +MOVJ EC01111
SMOVL C01112 +MOVJ EC01112
SMOVL C01113 +MOVJ EC01113
SMOVL C01114 +MOVJ EC01114
SMOVL C01115 +MOVJ EC01115
SMOVL C01116 +MOVJ EC01116
SMOVL C01117 +MOVJ EC01117
SMOVL C01118 +MOVJ EC01118
SMOVL C01119 +MOVJ EC01119
SMOVL C01120 +MOVJ EC01120
SMOVL C01121 +MOVJ EC01121
SMOVL C01122 +MOVJ EC01122
SMOVL C01123 +MOVJ EC01123
SMOVL C01124 +MOVJ EC01124
SMOVL C01125 +MOVJ EC01125
SMOVL C01126 +MOVJ EC01126
SMOVL C01127 +MOVJ EC01127
SMOVL C01128 +MOVJ EC01128
SMOVL C01129 +MOVJ EC01129
SMOVL C01130 +MOVJ EC01130
SMOVL C01131 +MOVJ EC01131
SMOVL C01132 +MOVJ EC01132
SMOVL C01133 +MOVJ EC01133
SMOVL C01134 +MOVJ EC01134
SMOVL C01135 +MOVJ EC01135
SMOVL C01136 +MOVJ EC01136
SMOVL C01137 +MOVJ EC01137
SMOVL C01138 +MOVJ EC01138
SMOVL C01139 +MOVJ EC01139
SMOVL C01140 +MOVJ EC01140
SMOVL C01141 +MOVJ EC01141
SMOVL C01142 +MOVJ EC01142
SMOVL C01143 +MOVJ EC01143
SMOVL C01144 +MOVJ EC01144
SMOVL C01145 +MOVJ EC01145
SMOVL C01146 +MOVJ EC01146
SMOVL C01147 +MOVJ EC01147
SMOVL C01148 +MOVJ EC01148
SMOVL C01149 +MOVJ EC01149
SMOVL C01150 +MOVJ EC01150
SMOVL C01151 +MOVJ EC01151
SMOVL C01152 +MOVJ EC01152
SMOVL C01153 +MOVJ EC01153
SMOVL C01154 +MOVJ EC01154
SMOVL C01155 +MOVJ EC01155
SMOVL C01156 +MOVJ EC01156
SMOVL C01157 +MOVJ EC01157
SMOVL C01158 +MOVJ EC01158
SMOVL C01159 +MOVJ EC01159
SMOVL C01160 +MOVJ EC01160
SMOVL C01161 +MOVJ EC01161
SMOVL C01162 +MOVJ EC01162
SMOVL C01163 +MOVJ EC01163
SMOVL C01164 +MOVJ EC01164
SMOVL C01165 +MOVJ EC01165
SMOVL C01166 +MOVJ EC01166
SMOVL C01167 +MOVJ EC01167
SMOVL C01168 +MOVJ EC01168
SMOVL C01169 +MOVJ EC01169
SMOVL C01170 +MOVJ EC01170
SMOVL C01171 +MOVJ EC01171
SMOVL C01172 +MOVJ EC01172
SMOVL C01173 +MOVJ EC01173
SMOVL C01174 +MOVJ EC01174
SMOVL C01175 +MOVJ EC01175
SMOVL C01176 +MOVJ EC01176
SMOVL C01177 +MOVJ EC01177
SMOVL C01178 +MOVJ EC01178
SMOVL C01179 +MOVJ EC01179
SMOVL C01180 +MOVJ EC01180
SMOVL C01181 +MOVJ EC01181
SMOVL C01182 +MOVJ EC01182
SMOVL C01183 +MOVJ EC01183
SMOVL C01184 +MOVJ EC01184
SMOVL C01185 +MOVJ EC01185
SMOVL C01186 +MOVJ EC01186
SMOVL C01187 +MOVJ EC01187
SMOVL C01188 +MOVJ EC01188
SMOVL C01189 +MOVJ EC01189
SMOVL C01190 +MOVJ EC01190
SMOVL C01191 +MOVJ EC01191
SMOVL C01192 +MOVJ EC01192
SMOVL C01193 +MOVJ EC01193
SMOVL C01194 +MOVJ EC01194
SMOVL C01195 +MOVJ EC01195
SMOVL C01196 +MOVJ EC01196
SMOVL C01197 +MOVJ EC01197
SMOVL C01198 +MOVJ EC01198
SMOVL C01199 +MOVJ EC01199
SMOVL C01200 +MOVJ EC01200
SMOVL C01201 +MOVJ EC01201
SMOVL C01202 +MOVJ EC01202
SMOVL C01203 +MOVJ EC01203
SMOVL C01204 +MOVJ EC01204
SMOVL C01205 +MOVJ EC01205
SMOVL C01206 +MOVJ EC01206
SMOVL C01207 +MOVJ EC01207
SMOVL C01208 +MOVJ EC01208
SMOVL C01209 +MOVJ EC01209
SMOVL C01210 +MOVJ EC01210
SMOVL C01211 +MOVJ EC01211
SMOVL C01212 +MOVJ EC01212
SMOVL C01213 +MOVJ EC01213
SMOVL C01214 +MOVJ EC01214
SMOVL C01215 +MOVJ EC01215
SMOVL C01216 +MOVJ EC01216
SMOVL C01217 +MOVJ EC01217
SMOVL C01218 +MOVJ EC01218
SMOVL C01219 +MOVJ EC01219
SMOVL C01220 +MOVJ EC01220
SMOVL C01221 +MOVJ EC01221
SMOVL C01222 +MOVJ EC01222
SMOVL C01223 +MOVJ EC01223
SMOVL C01224 +MOVJ EC01224
SMOVL C01225 +MOVJ EC01225
SMOVL C01226 +MOVJ EC01226
SMOVL C01227 +MOVJ EC01227
SMOVL C01228 +MOVJ EC01228
SMOVL C01229 +MOVJ EC01229
SMOVL C01230 +MOVJ EC01230
SMOVL C01231 +MOVJ EC01231
SMOVL C01232 +MOVJ EC01232
SMOVL C01233 +MOVJ EC01233
SMOVL C01234 +MOVJ EC01234
SMOVL C01235 +MOVJ EC01235
SMOVL C01236 +MOVJ EC01236
SMOVL C01237 +MOVJ EC01237
SMOVL C01238 +MOVJ EC01238
SMOVL C01239 +MOVJ EC01239
SMOVL C01240 +MOVJ EC01240
SMOVL C01241 +MOVJ EC01241
SMOVL C01242 +MOVJ EC01242
SMOVL C01243 +MOVJ EC01243
SMOVL C01244 +MOVJ EC01244
SMOVL C01245 +MOVJ EC01245
SMOVL C01246 +MOVJ EC01246
SMOVL C01247 +MOVJ EC01247
SMOVL C01248 +MOVJ EC01248
SMOVL C01249 +MOVJ EC01249
SMOVL C01250 +MOVJ EC01250
SMOVL C01251 +MOVJ EC01251
SMOVL C01252 +MOVJ EC01252
SMOVL C01253 +MOVJ EC01253
SMOVL C01254 +MOVJ EC01254
SMOVL C01255 +MOVJ EC01255
SMOVL C01256 +MOVJ EC01256
SMOVL C01257 +MOVJ EC01257
SMOVL C01258 +MOVJ EC01258
SMOVL C01259 +MOVJ EC01259
